LIN {X 0,Y 206.357,Z 449.351,A -85,B 0,C 180,E1 -22994.34,E2 -22994.34} C_VEL
LIN {X 0,Y 205.229,Z 439.622,A -85,B 0,C 180,E1 -22997.247,E2 -22997.247} C_VEL
LIN {X 0,Y 203.64,Z 431.973,A -85,B 0,C 180,E1 -22999.611,E2 -22999.611} C_VEL
LIN {X 0,Y 201.242,Z 425.032,A -85,B 0,C 180,E1 -23002.05,E2 -23002.05} C_VEL
LIN {X 0,Y 197.447,Z 417.118,A -85,B 0,C 180,E1 -23005.284,E2 -23005.284} C_VEL
LIN {X 0,Y 193.926,Z 410.394,A -85,B 0,C 180,E1 -23008.299,E2 -23008.299} C_VEL
LIN {X 0,Y 191.536,Z 406.308,A -85,B 0,C 180,E1 -23010.369,E2 -23010.369} C_VEL
LIN {X 0,Y 189.131,Z 402.897,A -85,B 0,C 180,E1 -23012.398,E2 -23012.398} C_VEL
LIN {X 0,Y 188.252,Z 401.374,A -85,B 0,C 180,E1 -23013.235,E2 -23013.235} C_VEL
LIN {X 0,Y 185.97,Z 398.361,A -85,B 0,C 180,E1 -23015.354,E2 -23015.354} C_VEL
LIN {X 0,Y 185.027,Z 396.629,A -85,B 0,C 180,E1 -23016.346,E2 -23016.346} C_VEL
LIN {X 0,Y 182.514,Z 394.01,A -85,B 0,C 180,E1 -23018.838,E2 -23018.838} C_VEL
LIN {X 0,Y 181.303,Z 391.376,A -85,B 0,C 180,E1 -23020.467,E2 -23020.467} C_VEL
LIN {X 0,Y 178.541,Z 389.25,A -85,B 0,C 180,E1 -23023.712,E2 -23023.712} C_VEL
LIN {X 0,Y 177.229,Z 386.47,A -85,B 0,C 180,E1 -23026.016,E2 -23026.016} C_VEL
LIN {X 0,Y 177.02,Z 385.707,A -85,B 0,C 180,E1 -23026.511,E2 -23026.511} C_VEL
LIN {X 0,Y 172.999,Z 381.886,A -85,B 0,C 180,E1 -23040,E2 -23040} C_VEL
LIN {X 0,Y 174.879,Z 384.888,A -85,B 0,C 180,E1 -23048.959,E2 -23048.959} C_VEL
LIN {X 0,Y 177.427,Z 387.578,A -85,B 0,C 180,E1 -23053.602,E2 -23053.602} C_VEL
LIN {X 0,Y 179.019,Z 391.368,A -85,B 0,C 180,E1 -23056.243,E2 -23056.243} C_VEL
LIN {X 0,Y 181.998,Z 394.906,A -85,B 0,C 180,E1 -23059.748,E2 -23059.748} C_VEL
LIN {X 0,Y 183.712,Z 398.579,A -85,B 0,C 180,E1 -23061.752,E2 -23061.752} C_VEL
LIN {X 0,Y 185.943,Z 401.558,A -85,B 0,C 180,E1 -23063.899,E2 -23063.899} C_VEL
LIN {X 0,Y 187.812,Z 405.564,A -85,B 0,C 180,E1 -23065.786,E2 -23065.786} C_VEL
LIN {X 0,Y 189.272,Z 407.823,A -85,B 0,C 180,E1 -23067.048,E2 -23067.048} C_VEL
LIN {X 0,Y 191.444,Z 412.238,A -85,B 0,C 180,E1 -23069.03,E2 -23069.03} C_VEL
LIN {X 0,Y 194.937,Z 419.942,A -85,B 0,C 180,E1 -23072.125,E2 -23072.125} C_VEL
LIN {X 0,Y 197.223,Z 425.43,A -85,B 0,C 180,E1 -23074.142,E2 -23074.142} C_VEL
LIN {X 0,Y 200.62,Z 435.333,A -85,B 0,C 180,E1 -23077.407,E2 -23077.407} C_VEL
LIN {X 0,Y 201.683,Z 440.477,A -85,B 0,C 180,E1 -23078.847,E2 -23078.847} C_VEL
LIN {X 0,Y 202.508,Z 450.041,A -85,B 0,C 180,E1 -23081.253,E2 -23081.253} C_VEL
LIN {X 0,Y 202.585,Z 459.199,A -85,B 0,C 180,E1 -23083.502,E2 -23083.502} C_VEL
LIN {X 0,Y 201.927,Z 468.704,A -85,B 0,C 180,E1 -23085.887,E2 -23085.887} C_VEL
LIN {X 0,Y 200.829,Z 476.69,A -85,B 0,C 180,E1 -23087.965,E2 -23087.965} C_VEL
LIN {X 0,Y 195.602,Z 487.568,A -85,B 0,C 180,E1 -23090.376,E2 -23090.376} C_VEL
LIN {X 0,Y 190.484,Z 497.578,A -85,B 0,C 180,E1 -23093.163,E2 -23093.163} C_VEL
LIN {X 0,Y 185.183,Z 507.379,A -85,B 0,C 180,E1 -23096.609,E2 -23096.609} C_VEL
LIN {X 0,Y 180.687,Z 515.593,A -85,B 0,C 180,E1 -23100.271,E2 -23100.271} C_VEL
LIN {X 0,Y 176.716,Z 522.382,A -85,B 0,C 180,E1 -23104.059,E2 -23104.059} C_VEL
LIN {X 0,Y 173.038,Z 529.281,A -85,B 0,C 180,E1 -23109.091,E2 -23109.091} C_VEL
LIN {X 0,Y 170.943,Z 533.56,A -85,B 0,C 180,E1 -23113.275,E2 -23113.275} C_VEL
LIN {X 0,Y 169.503,Z 537.155,A -85,B 0,C 180,E1 -23118.036,E2 -23118.036} C_VEL
LIN {X 0,Y 169.009,Z 539.54,A -85,B 0,C 180,E1 -23122.835,E2 -23122.835} C_VEL
LIN {X 0,Y 169.061,Z 540.479,A -85,B 0,C 180,E1 -23126.109,E2 -23126.109} C_VEL
LIN {X 0,Y 169.248,Z 540.917,A -85,B 0,C 180,E1 -23130.001,E2 -23130.001} C_VEL
LIN {X 0,Y 169.056,Z 540.278,A -85,B 0,C 180,E1 -23134.77,E2 -23134.77} C_VEL
LIN {X 0,Y 169.154,Z 538.458,A -85,B 0,C 180,E1 -23139.567,E2 -23139.567} C_VEL
LIN {X 0,Y 169.375,Z 537.495,A -85,B 0,C 180,E1 -23141.282,E2 -23141.282} C_VEL
LIN {X 0,Y 169.115,Z 536.308,A -85,B 0,C 180,E1 -23143.24,E2 -23143.24} C_VEL
LIN {X 0,Y 167.216,Z 533.952,A -85,B 0,C 180,E1 -23146.464,E2 -23146.464} C_VEL
LIN {X 0,Y 165.895,Z 531.695,A -85,B 0,C 180,E1 -23149.055,E2 -23149.055} C_VEL
LIN {X 0,Y 165.906,Z 529.739,A -85,B 0,C 180,E1 -23150.989,E2 -23150.989} C_VEL
LIN {X 0,Y 166.215,Z 529.037,A -85,B 0,C 180,E1 -23151.617,E2 -23151.617} C_VEL
LIN {X 0,Y 169.271,Z 523.624,A -85,B 0,C 180,E1 -23155.847,E2 -23155.847} C_VEL
LIN {X 0,Y 173.849,Z 516.138,A -85,B 0,C 180,E1 -23160.354,E2 -23160.354} C_VEL
LIN {X 0,Y 177.837,Z 509.382,A -85,B 0,C 180,E1 -23163.593,E2 -23163.593} C_VEL
LIN {X 0,Y 183.114,Z 500.046,A -85,B 0,C 180,E1 -23167.193,E2 -23167.193} C_VEL
LIN {X 0,Y 188.347,Z 490.582,A -85,B 0,C 180,E1 -23170.067,E2 -23170.067} C_VEL
LIN {X 0,Y 194.056,Z 479.351,A -85,B 0,C 180,E1 -23172.771,E2 -23172.771} C_VEL
LIN {X 0,Y 195.076,Z 476.407,A -85,B 0,C 180,E1 -23173.465,E2 -23173.465} C_VEL
LIN {X 0,Y 196.535,Z 465.476,A -85,B 0,C 180,E1 -23176.42,E2 -23176.42} C_VEL
LIN {X 0,Y 197.004,Z 454.416,A -85,B 0,C 180,E1 -23179.295,E2 -23179.295} C_VEL
LIN {X 0,Y 196.407,Z 443.528,A -85,B 0,C 180,E1 -23182.193,E2 -23182.193} C_VEL
LIN {X 0,Y 195.356,Z 438.125,A -85,B 0,C 180,E1 -23183.845,E2 -23183.845} C_VEL
LIN {X 0,Y 192.243,Z 428.566,A -85,B 0,C 180,E1 -23187.229,E2 -23187.229} C_VEL
LIN {X 0,Y 189.538,Z 421.776,A -85,B 0,C 180,E1 -23189.962,E2 -23189.962} C_VEL
LIN {X 0,Y 187.417,Z 417.073,A -85,B 0,C 180,E1 -23192.048,E2 -23192.048} C_VEL
LIN {X 0,Y 185.403,Z 412.52,A -85,B 0,C 180,E1 -23194.177,E2 -23194.177} C_VEL
LIN {X 0,Y 183.355,Z 408.488,A -85,B 0,C 180,E1 -23196.343,E2 -23196.343} C_VEL
LIN {X 0,Y 182.725,Z 407.139,A -85,B 0,C 180,E1 -23197.081,E2 -23197.081} C_VEL
LIN {X 0,Y 180.343,Z 403.371,A -85,B 0,C 180,E1 -23199.706,E2 -23199.706} C_VEL
LIN {X 0,Y 179.32,Z 400.892,A -85,B 0,C 180,E1 -23201.135,E2 -23201.135} C_VEL
LIN {X 0,Y 176.635,Z 397.089,A -85,B 0,C 180,E1 -23204.79,E2 -23204.79} C_VEL
LIN {X 0,Y 175.579,Z 394.08,A -85,B 0,C 180,E1 -23206.841,E2 -23206.841} C_VEL
LIN {X 0,Y 172.61,Z 390.708,A -85,B 0,C 180,E1 -23213.278,E2 -23213.278} C_VEL
LIN {X 0,Y 171.67,Z 388.393,A -85,B 0,C 180,E1 -23220,E2 -23220} C_VEL
LIN {X 0,Y 175.323,Z 392.776,A -85,B 0,C 180,E1 -23233.585,E2 -23233.585} C_VEL
LIN {X 0,Y 176.409,Z 395.611,A -85,B 0,C 180,E1 -23235.896,E2 -23235.896} C_VEL
LIN {X 0,Y 178.925,Z 397.987,A -85,B 0,C 180,E1 -23239.207,E2 -23239.207} C_VEL
LIN {X 0,Y 181.096,Z 401.825,A -85,B 0,C 180,E1 -23242.084,E2 -23242.084} C_VEL
LIN {X 0,Y 182.75,Z 403.698,A -85,B 0,C 180,E1 -23243.816,E2 -23243.816} C_VEL
LIN {X 0,Y 185.765,Z 408.54,A -85,B 0,C 180,E1 -23247,E2 -23247} C_VEL
LIN {X 0,Y 188.461,Z 413.028,A -85,B 0,C 180,E1 -23249.612,E2 -23249.612} C_VEL
LIN {X 0,Y 192.28,Z 420.206,A -85,B 0,C 180,E1 -23253.248,E2 -23253.248} C_VEL
LIN {X 0,Y 196.021,Z 428.537,A -85,B 0,C 180,E1 -23256.909,E2 -23256.909} C_VEL
LIN {X 0,Y 198.377,Z 435.704,A -85,B 0,C 180,E1 -23259.621,E2 -23259.621} C_VEL
LIN {X 0,Y 199.887,Z 444.192,A -85,B 0,C 180,E1 -23262.407,E2 -23262.407} C_VEL
LIN {X 0,Y 200.624,Z 454.153,A -85,B 0,C 180,E1 -23265.523,E2 -23265.523} C_VEL
LIN {X 0,Y 200.457,Z 456.426,A -85,B 0,C 180,E1 -23266.176,E2 -23266.176} C_VEL
LIN {X 0,Y 195.569,Z 467.034,A -85,B 0,C 180,E1 -23268.331,E2 -23268.331} C_VEL
LIN {X 0,Y 190.126,Z 477.796,A -85,B 0,C 180,E1 -23271.066,E2 -23271.066} C_VEL
LIN {X 0,Y 185.207,Z 486.911,A -85,B 0,C 180,E1 -23273.971,E2 -23273.971} C_VEL
LIN {X 0,Y 179.891,Z 495.825,A -85,B 0,C 180,E1 -23277.507,E2 -23277.507} C_VEL
LIN {X 0,Y 175.25,Z 503.202,A -85,B 0,C 180,E1 -23281.233,E2 -23281.233} C_VEL
LIN {X 0,Y 170.88,Z 510.082,A -85,B 0,C 180,E1 -23285.714,E2 -23285.714} C_VEL
LIN {X 0,Y 167.33,Z 515.481,A -85,B 0,C 180,E1 -23290.365,E2 -23290.365} C_VEL
LIN {X 0,Y 164.88,Z 519.538,A -85,B 0,C 180,E1 -23295.181,E2 -23295.181} C_VEL
LIN {X 0,Y 163.213,Z 522.382,A -85,B 0,C 180,E1 -23300.081,E2 -23300.081} C_VEL
LIN {X 0,Y 162.448,Z 524.08,A -85,B 0,C 180,E1 -23305.035,E2 -23305.035} C_VEL
LIN {X 0,Y 162.264,Z 524.667,A -85,B 0,C 180,E1 -23309.999,E2 -23309.999} C_VEL
LIN {X 0,Y 162.431,Z 524.114,A -85,B 0,C 180,E1 -23314.963,E2 -23314.963} C_VEL
LIN {X 0,Y 163.21,Z 522.46,A -85,B 0,C 180,E1 -23319.917,E2 -23319.917} C_VEL
LIN {X 0,Y 164.838,Z 519.657,A -85,B 0,C 180,E1 -23324.821,E2 -23324.821} C_VEL
LIN {X 0,Y 167.276,Z 515.639,A -85,B 0,C 180,E1 -23329.639,E2 -23329.639} C_VEL
LIN {X 0,Y 170.797,Z 510.291,A -85,B 0,C 180,E1 -23334.297,E2 -23334.297} C_VEL
LIN {X 0,Y 173.967,Z 505.297,A -85,B 0,C 180,E1 -23337.682,E2 -23337.682} C_VEL
LIN {X 0,Y 178.452,Z 498.328,A -85,B 0,C 180,E1 -23341.454,E2 -23341.454} C_VEL
LIN {X 0,Y 183.49,Z 489.94,A -85,B 0,C 180,E1 -23345.065,E2 -23345.065} C_VEL
LIN {X 0,Y 189.161,Z 479.921,A -85,B 0,C 180,E1 -23348.443,E2 -23348.443} C_VEL
LIN {X 0,Y 193.577,Z 471.337,A -85,B 0,C 180,E1 -23350.805,E2 -23350.805} C_VEL
LIN {X 0,Y 199.392,Z 459.291,A -85,B 0,C 180,E1 -23353.417,E2 -23353.417} C_VEL
LIN {X 0,Y 200.718,Z 455.857,A -85,B 0,C 180,E1 -23354.098,E2 -23354.098} C_VEL
LIN {X 0,Y 200.295,Z 447.148,A -85,B 0,C 180,E1 -23356.827,E2 -23356.827} C_VEL
LIN {X 0,Y 198.949,Z 437.956,A -85,B 0,C 180,E1 -23359.788,E2 -23359.788} C_VEL
LIN {X 0,Y 197.316,Z 431.708,A -85,B 0,C 180,E1 -23362.001,E2 -23362.001} C_VEL
LIN {X 0,Y 194.078,Z 424.015,A -85,B 0,C 180,E1 -23365.226,E2 -23365.226} C_VEL
LIN {X 0,Y 190.313,Z 416.234,A -85,B 0,C 180,E1 -23368.868,E2 -23368.868} C_VEL
LIN {X 0,Y 188.189,Z 412.289,A -85,B 0,C 180,E1 -23370.955,E2 -23370.955} C_VEL
LIN {X 0,Y 182.602,Z 403.311,A -85,B 0,C 180,E1 -23376.69,E2 -23376.69} C_VEL
LIN {X 0,Y 179.966,Z 400.122,A -85,B 0,C 180,E1 -23379.664,E2 -23379.664} C_VEL
LIN {X 0,Y 179.04,Z 398.02,A -85,B 0,C 180,E1 -23381.045,E2 -23381.045} C_VEL
LIN {X 0,Y 176.502,Z 395.71,A -85,B 0,C 180,E1 -23384.408,E2 -23384.408} C_VEL
LIN {X 0,Y 175.352,Z 392.774,A -85,B 0,C 180,E1 -23386.897,E2 -23386.897} C_VEL
LIN {X 0,Y 171.894,Z 388.908,A -85,B 0,C 180,E1 -23400,E2 -23400} C_VEL
LIN {X 0,Y 173.577,Z 391.852,A -85,B 0,C 180,E1 -23408.733,E2 -23408.733} C_VEL
LIN {X 0,Y 175.707,Z 394.352,A -85,B 0,C 180,E1 -23413.002,E2 -23413.002} C_VEL
LIN {X 0,Y 177.14,Z 397.978,A -85,B 0,C 180,E1 -23415.681,E2 -23415.681} C_VEL
LIN {X 0,Y 179.687,Z 401.392,A -85,B 0,C 180,E1 -23419.047,E2 -23419.047} C_VEL
LIN {X 0,Y 181.35,Z 405.086,A -85,B 0,C 180,E1 -23421.229,E2 -23421.229} C_VEL
LIN {X 0,Y 183.161,Z 407.746,A -85,B 0,C 180,E1 -23423.16,E2 -23423.16} C_VEL
LIN {X 0,Y 185.034,Z 411.929,A -85,B 0,C 180,E1 -23425.296,E2 -23425.296} C_VEL
LIN {X 0,Y 186.069,Z 413.773,A -85,B 0,C 180,E1 -23426.302,E2 -23426.302} C_VEL
LIN {X 0,Y 188.643,Z 419.492,A -85,B 0,C 180,E1 -23428.968,E2 -23428.968} C_VEL
LIN {X 0,Y 192.315,Z 428.597,A -85,B 0,C 180,E1 -23432.68,E2 -23432.68} C_VEL
LIN {X 0,Y 195.584,Z 438.822,A -85,B 0,C 180,E1 -23436.293,E2 -23436.293} C_VEL
LIN {X 0,Y 196.691,Z 445.183,A -85,B 0,C 180,E1 -23438.18,E2 -23438.18} C_VEL
LIN {X 0,Y 197.085,Z 455.509,A -85,B 0,C 180,E1 -23440.925,E2 -23440.925} C_VEL
LIN {X 0,Y 196.495,Z 467.003,A -85,B 0,C 180,E1 -23443.929,E2 -23443.929} C_VEL
LIN {X 0,Y 194.961,Z 477.492,A -85,B 0,C 180,E1 -23446.772,E2 -23446.772} C_VEL
LIN {X 0,Y 189.232,Z 489.017,A -85,B 0,C 180,E1 -23449.464,E2 -23449.464} C_VEL
LIN {X 0,Y 183.939,Z 498.727,A -85,B 0,C 180,E1 -23452.315,E2 -23452.315} C_VEL
LIN {X 0,Y 178.827,Z 507.692,A -85,B 0,C 180,E1 -23455.62,E2 -23455.62} C_VEL
LIN {X 0,Y 173.865,Z 516.266,A -85,B 0,C 180,E1 -23459.651,E2 -23459.651} C_VEL
LIN {X 0,Y 169.271,Z 523.722,A -85,B 0,C 180,E1 -23464.155,E2 -23464.155} C_VEL
LIN {X 0,Y 166.142,Z 529.276,A -85,B 0,C 180,E1 -23468.532,E2 -23468.532} C_VEL
LIN {X 0,Y 164.064,Z 533.208,A -85,B 0,C 180,E1 -23472.552,E2 -23472.552} C_VEL
LIN {X 0,Y 162.498,Z 536.804,A -85,B 0,C 180,E1 -23477.512,E2 -23477.512} C_VEL
LIN {X 0,Y 161.924,Z 539.19,A -85,B 0,C 180,E1 -23482.519,E2 -23482.519} C_VEL
LIN {X 0,Y 161.964,Z 540.222,A -85,B 0,C 180,E1 -23486.393,E2 -23486.393} C_VEL
LIN {X 0,Y 162.167,Z 540.57,A -85,B 0,C 180,E1 -23490.001,E2 -23490.001} C_VEL
LIN {X 0,Y 161.946,Z 539.928,A -85,B 0,C 180,E1 -23494.98,E2 -23494.98} C_VEL
LIN {X 0,Y 162.107,Z 538.107,A -85,B 0,C 180,E1 -23499.988,E2 -23499.988} C_VEL
LIN {X 0,Y 163.137,Z 535.106,A -85,B 0,C 180,E1 -23504.981,E2 -23504.981} C_VEL
LIN {X 0,Y 165.255,Z 530.865,A -85,B 0,C 180,E1 -23509.892,E2 -23509.892} C_VEL
LIN {X 0,Y 166.215,Z 529.037,A -85,B 0,C 180,E1 -23511.617,E2 -23511.617} C_VEL
LIN {X 0,Y 166.827,Z 526.887,A -85,B 0,C 180,E1 -23513.493,E2 -23513.493} C_VEL
LIN {X 0,Y 166.204,Z 519.756,A -85,B 0,C 180,E1 -23519.123,E2 -23519.123} C_VEL
LIN {X 0,Y 166.985,Z 517.012,A -85,B 0,C 180,E1 -23520.904,E2 -23520.904} C_VEL
LIN {X 0,Y 167.525,Z 516.025,A -85,B 0,C 180,E1 -23521.462,E2 -23521.462} C_VEL
LIN {X 0,Y 172.577,Z 507.794,A -85,B 0,C 180,E1 -23525.465,E2 -23525.465} C_VEL
LIN {X 0,Y 178.346,Z 498.194,A -85,B 0,C 180,E1 -23529.089,E2 -23529.089} C_VEL
LIN {X 0,Y 183.836,Z 488.443,A -85,B 0,C 180,E1 -23531.993,E2 -23531.993} C_VEL
LIN {X 0,Y 188.881,Z 478.998,A -85,B 0,C 180,E1 -23534.241,E2 -23534.241} C_VEL
LIN {X 0,Y 190.432,Z 470.051,A -85,B 0,C 180,E1 -23536.793,E2 -23536.793} C_VEL
LIN {X 0,Y 191.405,Z 460.211,A -85,B 0,C 180,E1 -23539.513,E2 -23539.513} C_VEL
LIN {X 0,Y 191.437,Z 449.894,A -85,B 0,C 180,E1 -23542.387,E2 -23542.387} C_VEL
LIN {X 0,Y 190.929,Z 444.234,A -85,B 0,C 180,E1 -23544.079,E2 -23544.079} C_VEL
LIN {X 0,Y 188.11,Z 434.077,A -85,B 0,C 180,E1 -23547.817,E2 -23547.817} C_VEL
LIN {X 0,Y 185.33,Z 426.351,A -85,B 0,C 180,E1 -23551.086,E2 -23551.086} C_VEL
LIN {X 0,Y 182.601,Z 419.461,A -85,B 0,C 180,E1 -23554.343,E2 -23554.343} C_VEL
LIN {X 0,Y 179.328,Z 412.591,A -85,B 0,C 180,E1 -23558.333,E2 -23558.333} C_VEL
LIN {X 0,Y 177.226,Z 408.252,A -85,B 0,C 180,E1 -23561.204,E2 -23561.204} C_VEL
LIN {X 0,Y 176.746,Z 407.099,A -85,B 0,C 180,E1 -23561.977,E2 -23561.977} C_VEL
LIN {X 0,Y 174.423,Z 403.409,A -85,B 0,C 180,E1 -23565.554,E2 -23565.554} C_VEL
LIN {X 0,Y 173.633,Z 400.759,A -85,B 0,C 180,E1 -23567.435,E2 -23567.435} C_VEL
LIN {X 0,Y 171.059,Z 397.556,A -85,B 0,C 180,E1 -23573.661,E2 -23573.661} C_VEL
LIN {X 0,Y 170.307,Z 395.372,A -85,B 0,C 180,E1 -23580,E2 -23580} C_VEL
LIN {X 0,Y 173.338,Z 399.597,A -85,B 0,C 180,E1 -23593.115,E2 -23593.115} C_VEL
LIN {X 0,Y 174.397,Z 402.424,A -85,B 0,C 180,E1 -23595.635,E2 -23595.635} C_VEL
LIN {X 0,Y 176.681,Z 404.826,A -85,B 0,C 180,E1 -23598.955,E2 -23598.955} C_VEL
LIN {X 0,Y 177.884,Z 407.4,A -85,B 0,C 180,E1 -23600.829,E2 -23600.829} C_VEL
LIN {X 0,Y 179.705,Z 409.616,A -85,B 0,C 180,E1 -23603.022,E2 -23603.022} C_VEL
LIN {X 0,Y 182.445,Z 414.39,A -85,B 0,C 180,E1 -23606.295,E2 -23606.295} C_VEL
LIN {X 0,Y 185.331,Z 419.821,A -85,B 0,C 180,E1 -23609.537,E2 -23609.537} C_VEL
LIN {X 0,Y 188.386,Z 426.072,A -85,B 0,C 180,E1 -23612.839,E2 -23612.839} C_VEL
LIN {X 0,Y 191.66,Z 434.084,A -85,B 0,C 180,E1 -23616.509,E2 -23616.509} C_VEL
LIN {X 0,Y 193.437,Z 440.358,A -85,B 0,C 180,E1 -23618.992,E2 -23618.992} C_VEL
LIN {X 0,Y 194.566,Z 448.821,A -85,B 0,C 180,E1 -23621.932,E2 -23621.932} C_VEL
LIN {X 0,Y 194.864,Z 458.05,A -85,B 0,C 180,E1 -23624.977,E2 -23624.977} C_VEL
LIN {X 0,Y 189.36,Z 469.319,A -85,B 0,C 180,E1 -23627.363,E2 -23627.363} C_VEL
LIN {X 0,Y 184.633,Z 478.149,A -85,B 0,C 180,E1 -23629.675,E2 -23629.675} C_VEL
LIN {X 0,Y 179.507,Z 487.261,A -85,B 0,C 180,E1 -23632.637,E2 -23632.637} C_VEL
LIN {X 0,Y 173.941,Z 496.175,A -85,B 0,C 180,E1 -23636.249,E2 -23636.249} C_VEL
LIN {X 0,Y 169.059,Z 503.552,A -85,B 0,C 180,E1 -23640.075,E2 -23640.075} C_VEL
LIN {X 0,Y 164.39,Z 510.433,A -85,B 0,C 180,E1 -23644.689,E2 -23644.689} C_VEL
LIN {X 0,Y 160.641,Z 515.831,A -85,B 0,C 180,E1 -23649.512,E2 -23649.512} C_VEL
LIN {X 0,Y 158.001,Z 519.888,A -85,B 0,C 180,E1 -23654.52,E2 -23654.52} C_VEL
LIN {X 0,Y 156.234,Z 522.73,A -85,B 0,C 180,E1 -23659.633,E2 -23659.633} C_VEL
LIN {X 0,Y 155.383,Z 524.427,A -85,B 0,C 180,E1 -23664.809,E2 -23664.809} C_VEL
LIN {X 0,Y 155.187,Z 525.014,A -85,B 0,C 180,E1 -23669.999,E2 -23669.999} C_VEL
LIN {X 0,Y 155.473,Z 524.299,A -85,B 0,C 180,E1 -23676.015,E2 -23676.015} C_VEL
LIN {X 0,Y 156.229,Z 522.807,A -85,B 0,C 180,E1 -23680.365,E2 -23680.365} C_VEL
LIN {X 0,Y 157.962,Z 520.006,A -85,B 0,C 180,E1 -23685.482,E2 -23685.482} C_VEL
LIN {X 0,Y 160.586,Z 515.987,A -85,B 0,C 180,E1 -23690.493,E2 -23690.493} C_VEL
LIN {X 0,Y 164.297,Z 510.641,A -85,B 0,C 180,E1 -23695.324,E2 -23695.324} C_VEL
LIN {X 0,Y 168.968,Z 503.817,A -85,B 0,C 180,E1 -23699.941,E2 -23699.941} C_VEL
LIN {X 0,Y 173.858,Z 496.471,A -85,B 0,C 180,E1 -23703.767,E2 -23703.767} C_VEL
LIN {X 0,Y 179.384,Z 487.606,A -85,B 0,C 180,E1 -23707.391,E2 -23707.391} C_VEL
LIN {X 0,Y 184.809,Z 478.087,A -85,B 0,C 180,E1 -23710.485,E2 -23710.485} C_VEL
LIN {X 0,Y 190.215,Z 467.874,A -85,B 0,C 180,E1 -23713.119,E2 -23713.119} C_VEL
LIN {X 0,Y 194.774,Z 458.524,A -85,B 0,C 180,E1 -23715.081,E2 -23715.081} C_VEL
LIN {X 0,Y 194.957,Z 455.123,A -85,B 0,C 180,E1 -23716.134,E2 -23716.134} C_VEL
LIN {X 0,Y 194.521,Z 447.32,A -85,B 0,C 180,E1 -23718.748,E2 -23718.748} C_VEL
LIN {X 0,Y 193.512,Z 440.125,A -85,B 0,C 180,E1 -23721.25,E2 -23721.25} C_VEL
LIN {X 0,Y 191.645,Z 433.849,A -85,B 0,C 180,E1 -23723.781,E2 -23723.781} C_VEL
LIN {X 0,Y 188.336,Z 425.795,A -85,B 0,C 180,E1 -23727.494,E2 -23727.494} C_VEL
LIN {X 0,Y 184.709,Z 418.303,A -85,B 0,C 180,E1 -23731.477,E2 -23731.477} C_VEL
LIN {X 0,Y 179.918,Z 410.036,A -85,B 0,C 180,E1 -23737.007,E2 -23737.007} C_VEL
LIN {X 0,Y 177.081,Z 405.761,A -85,B 0,C 180,E1 -23740.75,E2 -23740.75} C_VEL
LIN {X 0,Y 176.487,Z 404.509,A -85,B 0,C 180,E1 -23741.724,E2 -23741.724} C_VEL
LIN {X 0,Y 174.163,Z 401.948,A -85,B 0,C 180,E1 -23745.317,E2 -23745.317} C_VEL
LIN {X 0,Y 173.237,Z 399.316,A -85,B 0,C 180,E1 -23747.702,E2 -23747.702} C_VEL
LIN {X 0,Y 170.505,Z 395.884,A -85,B 0,C 180,E1 -23760,E2 -23760} C_VEL
LIN {X 0,Y 172.004,Z 398.75,A -85,B 0,C 180,E1 -23768.517,E2 -23768.517} C_VEL
LIN {X 0,Y 173.753,Z 401.032,A -85,B 0,C 180,E1 -23772.408,E2 -23772.408} C_VEL
LIN {X 0,Y 175.18,Z 404.84,A -85,B 0,C 180,E1 -23775.413,E2 -23775.413} C_VEL
LIN {X 0,Y 177.216,Z 407.877,A -85,B 0,C 180,E1 -23778.415,E2 -23778.415} C_VEL
LIN {X 0,Y 178.944,Z 411.83,A -85,B 0,C 180,E1 -23780.951,E2 -23780.951} C_VEL
LIN {X 0,Y 180.106,Z 413.513,A -85,B 0,C 180,E1 -23782.263,E2 -23782.263} C_VEL
LIN {X 0,Y 181.329,Z 416.899,A -85,B 0,C 180,E1 -23784.014,E2 -23784.014} C_VEL
LIN {X 0,Y 182.745,Z 419.751,A -85,B 0,C 180,E1 -23785.636,E2 -23785.636} C_VEL
LIN {X 0,Y 185.022,Z 425.348,A -85,B 0,C 180,E1 -23788.347,E2 -23788.347} C_VEL
LIN {X 0,Y 187.793,Z 432.86,A -85,B 0,C 180,E1 -23791.597,E2 -23791.597} C_VEL
LIN {X 0,Y 190.354,Z 441.59,A -85,B 0,C 180,E1 -23794.91,E2 -23794.91} C_VEL
LIN {X 0,Y 191.353,Z 446.787,A -85,B 0,C 180,E1 -23796.643,E2 -23796.643} C_VEL
LIN {X 0,Y 191.618,Z 455.971,A -85,B 0,C 180,E1 -23799.248,E2 -23799.248} C_VEL
LIN {X 0,Y 191.217,Z 463.853,A -85,B 0,C 180,E1 -23801.42,E2 -23801.42} C_VEL
LIN {X 0,Y 189.973,Z 473.824,A -85,B 0,C 180,E1 -23804.214,E2 -23804.214} C_VEL
LIN {X 0,Y 188.896,Z 479.242,A -85,B 0,C 180,E1 -23805.766,E2 -23805.766} C_VEL
LIN {X 0,Y 182.905,Z 490.439,A -85,B 0,C 180,E1 -23808.486,E2 -23808.486} C_VEL
LIN {X 0,Y 176.582,Z 501.319,A -85,B 0,C 180,E1 -23811.911,E2 -23811.911} C_VEL
LIN {X 0,Y 171.15,Z 510.407,A -85,B 0,C 180,E1 -23815.625,E2 -23815.625} C_VEL
LIN {X 0,Y 166.37,Z 517.957,A -85,B 0,C 180,E1 -23819.542,E2 -23819.542} C_VEL
LIN {X 0,Y 161.834,Z 525.012,A -85,B 0,C 180,E1 -23824.262,E2 -23824.262} C_VEL
LIN {X 0,Y 158.495,Z 530.582,A -85,B 0,C 180,E1 -23829.224,E2 -23829.224} C_VEL
LIN {X 0,Y 156.226,Z 534.81,A -85,B 0,C 180,E1 -23834.342,E2 -23834.342} C_VEL
LIN {X 0,Y 155.041,Z 537.794,A -85,B 0,C 180,E1 -23839.554,E2 -23839.554} C_VEL
LIN {X 0,Y 154.846,Z 539.595,A -85,B 0,C 180,E1 -23844.793,E2 -23844.793} C_VEL
LIN {X 0,Y 155.067,Z 540.222,A -85,B 0,C 180,E1 -23850.001,E2 -23850.001} C_VEL
LIN {X 0,Y 154.848,Z 539.578,A -85,B 0,C 180,E1 -23855.209,E2 -23855.209} C_VEL
LIN {X 0,Y 155.08,Z 537.757,A -85,B 0,C 180,E1 -23860.445,E2 -23860.445} C_VEL
LIN {X 0,Y 156.23,Z 534.754,A -85,B 0,C 180,E1 -23865.66,E2 -23865.66} C_VEL
LIN {X 0,Y 158.513,Z 530.512,A -85,B 0,C 180,E1 -23870.776,E2 -23870.776} C_VEL
LIN {X 0,Y 161.836,Z 524.915,A -85,B 0,C 180,E1 -23875.74,E2 -23875.74} C_VEL
LIN {X 0,Y 166.36,Z 517.826,A -85,B 0,C 180,E1 -23880.462,E2 -23880.462} C_VEL
LIN {X 0,Y 167.525,Z 516.025,A -85,B 0,C 180,E1 -23881.462,E2 -23881.462} C_VEL
LIN {X 0,Y 168.808,Z 513.064,A -85,B 0,C 180,E1 -23883.151,E2 -23883.151} C_VEL
LIN {X 0,Y 169.476,Z 508.033,A -85,B 0,C 180,E1 -23886.044,E2 -23886.044} C_VEL
LIN {X 0,Y 170.473,Z 502.549,A -85,B 0,C 180,E1 -23888.805,E2 -23888.805} C_VEL
LIN {X 0,Y 172.2,Z 498.882,A -85,B 0,C 180,E1 -23890.236,E2 -23890.236} C_VEL
LIN {X 0,Y 178.579,Z 488.089,A -85,B 0,C 180,E1 -23893.53,E2 -23893.53} C_VEL
LIN {X 0,Y 183.148,Z 479.713,A -85,B 0,C 180,E1 -23895.583,E2 -23895.583} C_VEL
LIN {X 0,Y 185.063,Z 469.654,A -85,B 0,C 180,E1 -23898.595,E2 -23898.595} C_VEL
LIN {X 0,Y 186.126,Z 458.7,A -85,B 0,C 180,E1 -23901.809,E2 -23901.809} C_VEL
LIN {X 0,Y 186.115,Z 450.316,A -85,B 0,C 180,E1 -23904.322,E2 -23904.322} C_VEL
LIN {X 0,Y 185.318,Z 445.395,A -85,B 0,C 180,E1 -23906.076,E2 -23906.076} C_VEL
LIN {X 0,Y 183.162,Z 437.048,A -85,B 0,C 180,E1 -23909.442,E2 -23909.442} C_VEL
LIN {X 0,Y 180.314,Z 428.581,A -85,B 0,C 180,E1 -23913.371,E2 -23913.371} C_VEL
LIN {X 0,Y 178.706,Z 424.196,A -85,B 0,C 180,E1 -23915.611,E2 -23915.611} C_VEL
LIN {X 0,Y 176.317,Z 418.715,A -85,B 0,C 180,E1 -23918.977,E2 -23918.977} C_VEL
LIN {X 0,Y 174.82,Z 415.549,A -85,B 0,C 180,E1 -23921.24,E2 -23921.24} C_VEL
LIN {X 0,Y 174.285,Z 413.624,A -85,B 0,C 180,E1 -23922.396,E2 -23922.396} C_VEL
LIN {X 0,Y 172.099,Z 409.894,A -85,B 0,C 180,E1 -23926.119,E2 -23926.119} C_VEL
LIN {X 0,Y 171.375,Z 407.292,A -85,B 0,C 180,E1 -23928.168,E2 -23928.168} C_VEL
LIN {X 0,Y 169.237,Z 404.365,A -85,B 0,C 180,E1 -23934.041,E2 -23934.041} C_VEL
LIN {X 0,Y 168.643,Z 402.308,A -85,B 0,C 180,E1 -23940,E2 -23940} C_VEL
LIN {X 0,Y 171.102,Z 406.261,A -85,B 0,C 180,E1 -23952.604,E2 -23952.604} C_VEL
LIN {X 0,Y 171.64,Z 408.08,A -85,B 0,C 180,E1 -23954.222,E2 -23954.222} C_VEL
LIN {X 0,Y 174.187,Z 411.885,A -85,B 0,C 180,E1 -23958.831,E2 -23958.831} C_VEL
LIN {X 0,Y 176.494,Z 415.577,A -85,B 0,C 180,E1 -23962.228,E2 -23962.228} C_VEL
LIN {X 0,Y 178.939,Z 420.188,A -85,B 0,C 180,E1 -23965.597,E2 -23965.597} C_VEL
LIN {X 0,Y 182.473,Z 427.355,A -85,B 0,C 180,E1 -23970.046,E2 -23970.046} C_VEL
LIN {X 0,Y 185.964,Z 436.051,A -85,B 0,C 180,E1 -23974.534,E2 -23974.534} C_VEL
LIN {X 0,Y 187.598,Z 441.129,A -85,B 0,C 180,E1 -23976.828,E2 -23976.828} C_VEL
LIN {X 0,Y 188.689,Z 447.432,A -85,B 0,C 180,E1 -23979.286,E2 -23979.286} C_VEL
LIN {X 0,Y 189.182,Z 455.756,A -85,B 0,C 180,E1 -23982.289,E2 -23982.289} C_VEL
LIN {X 0,Y 189.071,Z 460.211,A -85,B 0,C 180,E1 -23983.817,E2 -23983.817} C_VEL
LIN {X 0,Y 183.204,Z 471.581,A -85,B 0,C 180,E1 -23986.328,E2 -23986.328} C_VEL
LIN {X 0,Y 178.003,Z 480.807,A -85,B 0,C 180,E1 -23988.924,E2 -23988.924} C_VEL
LIN {X 0,Y 172.148,Z 490.291,A -85,B 0,C 180,E1 -23992.237,E2 -23992.237} C_VEL
LIN {X 0,Y 166.549,Z 498.736,A -85,B 0,C 180,E1 -23996.004,E2 -23996.004} C_VEL
LIN {X 0,Y 161.585,Z 505.757,A -85,B 0,C 180,E1 -23999.987,E2 -23999.987} C_VEL
LIN {X 0,Y 156.932,Z 512.255,A -85,B 0,C 180,E1 -24004.82,E2 -24004.82} C_VEL
LIN {X 0,Y 153.199,Z 517.326,A -85,B 0,C 180,E1 -24009.874,E2 -24009.874} C_VEL
LIN {X 0,Y 151.156,Z 520.237,A -85,B 0,C 180,E1 -24013.8,E2 -24013.8} C_VEL
LIN {X 0,Y 149.24,Z 523.08,A -85,B 0,C 180,E1 -24019.141,E2 -24019.141} C_VEL
LIN {X 0,Y 148.325,Z 524.775,A -85,B 0,C 180,E1 -24024.561,E2 -24024.561} C_VEL
LIN {X 0,Y 148.112,Z 525.361,A -85,B 0,C 180,E1 -24029.999,E2 -24029.999} C_VEL
LIN {X 0,Y 148.369,Z 524.733,A -85,B 0,C 180,E1 -24035.88,E2 -24035.88} C_VEL
LIN {X 0,Y 149.233,Z 523.156,A -85,B 0,C 180,E1 -24040.857,E2 -24040.857} C_VEL
LIN {X 0,Y 151.117,Z 520.354,A -85,B 0,C 180,E1 -24046.202,E2 -24046.202} C_VEL
LIN {X 0,Y 153.938,Z 516.335,A -85,B 0,C 180,E1 -24051.421,E2 -24051.421} C_VEL
LIN {X 0,Y 157.871,Z 510.989,A -85,B 0,C 180,E1 -24056.433,E2 -24056.433} C_VEL
LIN {X 0,Y 162.839,Z 504.164,A -85,B 0,C 180,E1 -24061.191,E2 -24061.191} C_VEL
LIN {X 0,Y 168.781,Z 495.63,A -85,B 0,C 180,E1 -24065.657,E2 -24065.657} C_VEL
LIN {X 0,Y 174.717,Z 486.544,A -85,B 0,C 180,E1 -24069.311,E2 -24069.311} C_VEL
LIN {X 0,Y 180.124,Z 477.295,A -85,B 0,C 180,E1 -24072.302,E2 -24072.302} C_VEL
LIN {X 0,Y 186.169,Z 466.278,A -85,B 0,C 180,E1 -24075.057,E2 -24075.057} C_VEL
LIN {X 0,Y 189.006,Z 460.632,A -85,B 0,C 180,E1 -24076.238,E2 -24076.238} C_VEL
LIN {X 0,Y 189.293,Z 458.382,A -85,B 0,C 180,E1 -24076.951,E2 -24076.951} C_VEL
LIN {X 0,Y 189.106,Z 450.896,A -85,B 0,C 180,E1 -24079.594,E2 -24079.594} C_VEL
LIN {X 0,Y 188.402,Z 444.349,A -85,B 0,C 180,E1 -24082.01,E2 -24082.01} C_VEL
LIN {X 0,Y 186.982,Z 438.82,A -85,B 0,C 180,E1 -24084.367,E2 -24084.367} C_VEL
LIN {X 0,Y 183.967,Z 430.788,A -85,B 0,C 180,E1 -24088.312,E2 -24088.312} C_VEL
LIN {X 0,Y 180.904,Z 423.867,A -85,B 0,C 180,E1 -24092.212,E2 -24092.212} C_VEL
LIN {X 0,Y 177.428,Z 417.554,A -85,B 0,C 180,E1 -24096.665,E2 -24096.665} C_VEL
LIN {X 0,Y 176.701,Z 415.958,A -85,B 0,C 180,E1 -24097.799,E2 -24097.799} C_VEL
LIN {X 0,Y 173.794,Z 410.924,A -85,B 0,C 180,E1 -24102.344,E2 -24102.344} C_VEL
LIN {X 0,Y 171.85,Z 408.501,A -85,B 0,C 180,E1 -24105.796,E2 -24105.796} C_VEL
LIN {X 0,Y 171.07,Z 406.031,A -85,B 0,C 180,E1 -24108.146,E2 -24108.146} C_VEL
LIN {X 0,Y 168.832,Z 402.807,A -85,B 0,C 180,E1 -24120,E2 -24120} C_VEL
LIN {X 0,Y 170.163,Z 405.572,A -85,B 0,C 180,E1 -24128.311,E2 -24128.311} C_VEL
LIN {X 0,Y 171.571,Z 407.603,A -85,B 0,C 180,E1 -24131.818,E2 -24131.818} C_VEL
LIN {X 0,Y 172.862,Z 411.434,A -85,B 0,C 180,E1 -24135.012,E2 -24135.012} C_VEL
LIN {X 0,Y 174.451,Z 413.926,A -85,B 0,C 180,E1 -24137.586,E2 -24137.586} C_VEL
LIN {X 0,Y 175.707,Z 417.392,A -85,B 0,C 180,E1 -24139.876,E2 -24139.876} C_VEL
LIN {X 0,Y 176.538,Z 418.812,A -85,B 0,C 180,E1 -24140.995,E2 -24140.995} C_VEL
LIN {X 0,Y 179.236,Z 425.532,A -85,B 0,C 180,E1 -24144.93,E2 -24144.93} C_VEL
LIN {X 0,Y 181.244,Z 431.113,A -85,B 0,C 180,E1 -24147.73,E2 -24147.73} C_VEL
LIN {X 0,Y 184.042,Z 439.93,A -85,B 0,C 180,E1 -24151.673,E2 -24151.673} C_VEL
LIN {X 0,Y 185.981,Z 448.366,A -85,B 0,C 180,E1 -24154.944,E2 -24154.944} C_VEL
LIN {X 0,Y 186.319,Z 453.623,A -85,B 0,C 180,E1 -24156.622,E2 -24156.622} C_VEL
LIN {X 0,Y 185.883,Z 463.706,A -85,B 0,C 180,E1 -24159.6,E2 -24159.6} C_VEL
LIN {X 0,Y 184.526,Z 473.434,A -85,B 0,C 180,E1 -24162.446,E2 -24162.446} C_VEL
LIN {X 0,Y 183.214,Z 479.908,A -85,B 0,C 180,E1 -24164.418,E2 -24164.418} C_VEL
LIN {X 0,Y 177.598,Z 490.09,A -85,B 0,C 180,E1 -24166.952,E2 -24166.952} C_VEL
LIN {X 0,Y 170.993,Z 500.969,A -85,B 0,C 180,E1 -24170.428,E2 -24170.428} C_VEL
LIN {X 0,Y 165.255,Z 510.056,A -85,B 0,C 180,E1 -24174.215,E2 -24174.215} C_VEL
LIN {X 0,Y 160.25,Z 517.609,A -85,B 0,C 180,E1 -24178.247,E2 -24178.247} C_VEL
LIN {X 0,Y 155.381,Z 524.66,A -85,B 0,C 180,E1 -24183.109,E2 -24183.109} C_VEL
LIN {X 0,Y 151.795,Z 530.23,A -85,B 0,C 180,E1 -24188.261,E2 -24188.261} C_VEL
LIN {X 0,Y 149.346,Z 534.46,A -85,B 0,C 180,E1 -24193.601,E2 -24193.601} C_VEL
LIN {X 0,Y 148.009,Z 537.443,A -85,B 0,C 180,E1 -24199.052,E2 -24199.052} C_VEL
LIN {X 0,Y 147.736,Z 539.245,A -85,B 0,C 180,E1 -24204.542,E2 -24204.542} C_VEL
LIN {X 0,Y 147.823,Z 539.708,A -85,B 0,C 180,E1 -24207.276,E2 -24207.276} C_VEL
LIN {X 0,Y 147.971,Z 539.874,A -85,B 0,C 180,E1 -24210.001,E2 -24210.001} C_VEL
LIN {X 0,Y 147.818,Z 539.65,A -85,B 0,C 180,E1 -24213.201,E2 -24213.201} C_VEL
LIN {X 0,Y 147.776,Z 538.462,A -85,B 0,C 180,E1 -24218.204,E2 -24218.204} C_VEL
LIN {X 0,Y 148.518,Z 536.052,A -85,B 0,C 180,E1 -24223.687,E2 -24223.687} C_VEL
LIN {X 0,Y 150.424,Z 532.441,A -85,B 0,C 180,E1 -24229.091,E2 -24229.091} C_VEL
LIN {X 0,Y 153.457,Z 527.537,A -85,B 0,C 180,E1 -24234.343,E2 -24234.343} C_VEL
LIN {X 0,Y 157.614,Z 521.213,A -85,B 0,C 180,E1 -24239.374,E2 -24239.374} C_VEL
LIN {X 0,Y 162.305,Z 514.407,A -85,B 0,C 180,E1 -24243.512,E2 -24243.512} C_VEL
LIN {X 0,Y 167.431,Z 506.428,A -85,B 0,C 180,E1 -24247.341,E2 -24247.341} C_VEL
LIN {X 0,Y 172.2,Z 498.882,A -85,B 0,C 180,E1 -24250.236,E2 -24250.236} C_VEL
LIN {X 0,Y 174.135,Z 495.15,A -85,B 0,C 180,E1 -24251.578,E2 -24251.578} C_VEL
LIN {X 0,Y 176.011,Z 488.767,A -85,B 0,C 180,E1 -24253.964,E2 -24253.964} C_VEL
LIN {X 0,Y 178.091,Z 478.062,A -85,B 0,C 180,E1 -24257.792,E2 -24257.792} C_VEL
LIN {X 0,Y 179.778,Z 469.336,A -85,B 0,C 180,E1 -24260.512,E2 -24260.512} C_VEL
LIN {X 0,Y 180.778,Z 460.237,A -85,B 0,C 180,E1 -24263.334,E2 -24263.334} C_VEL
LIN {X 0,Y 180.896,Z 452.357,A -85,B 0,C 180,E1 -24265.896,E2 -24265.896} C_VEL
LIN {X 0,Y 179.033,Z 443.151,A -85,B 0,C 180,E1 -24269.727,E2 -24269.727} C_VEL
LIN {X 0,Y 176.774,Z 434.977,A -85,B 0,C 180,E1 -24273.596,E2 -24273.596} C_VEL
LIN {X 0,Y 175.116,Z 429.902,A -85,B 0,C 180,E1 -24276.339,E2 -24276.339} C_VEL
LIN {X 0,Y 173.01,Z 424.493,A -85,B 0,C 180,E1 -24279.801,E2 -24279.801} C_VEL
LIN {X 0,Y 171.253,Z 419.625,A -85,B 0,C 180,E1 -24283.306,E2 -24283.306} C_VEL
LIN {X 0,Y 169.493,Z 416.163,A -85,B 0,C 180,E1 -24286.818,E2 -24286.818} C_VEL
LIN {X 0,Y 169.143,Z 414.725,A -85,B 0,C 180,E1 -24288.01,E2 -24288.01} C_VEL
LIN {X 0,Y 168.317,Z 412.895,A -85,B 0,C 180,E1 -24290.386,E2 -24290.386} C_VEL
LIN {X 0,Y 166.991,Z 410.844,A -85,B 0,C 180,E1 -24295.172,E2 -24295.172} C_VEL
LIN {X 0,Y 166.686,Z 409.158,A -85,B 0,C 180,E1 -24300,E2 -24300} C_VEL
LIN {X 0,Y 168.643,Z 412.714,A -85,B 0,C 180,E1 -24312.027,E2 -24312.027} C_VEL
LIN {X 0,Y 169.36,Z 415.065,A -85,B 0,C 180,E1 -24314.418,E2 -24314.418} C_VEL
LIN {X 0,Y 171.073,Z 417.893,A -85,B 0,C 180,E1 -24317.946,E2 -24317.946} C_VEL
LIN {X 0,Y 173.117,Z 421.479,A -85,B 0,C 180,E1 -24321.431,E2 -24321.431} C_VEL
LIN {X 0,Y 175.235,Z 425.799,A -85,B 0,C 180,E1 -24324.832,E2 -24324.832} C_VEL
LIN {X 0,Y 178.044,Z 432.093,A -85,B 0,C 180,E1 -24328.982,E2 -24328.982} C_VEL
LIN {X 0,Y 180.757,Z 439.219,A -85,B 0,C 180,E1 -24332.979,E2 -24332.979} C_VEL
LIN {X 0,Y 182.604,Z 445.546,A -85,B 0,C 180,E1 -24336.074,E2 -24336.074} C_VEL
LIN {X 0,Y 183.417,Z 451.722,A -85,B 0,C 180,E1 -24338.624,E2 -24338.624} C_VEL
LIN {X 0,Y 183.595,Z 459.969,A -85,B 0,C 180,E1 -24341.751,E2 -24341.751} C_VEL
LIN {X 0,Y 183.149,Z 462.651,A -85,B 0,C 180,E1 -24342.656,E2 -24342.656} C_VEL
LIN {X 0,Y 177.082,Z 473.701,A -85,B 0,C 180,E1 -24345.213,E2 -24345.213} C_VEL
LIN {X 0,Y 171.864,Z 482.607,A -85,B 0,C 180,E1 -24347.835,E2 -24347.835} C_VEL
LIN {X 0,Y 165.715,Z 491.98,A -85,B 0,C 180,E1 -24351.276,E2 -24351.276} C_VEL
LIN {X 0,Y 159.906,Z 500.189,A -85,B 0,C 180,E1 -24355.154,E2 -24355.154} C_VEL
LIN {X 0,Y 154.104,Z 507.892,A -85,B 0,C 180,E1 -24359.889,E2 -24359.889} C_VEL
LIN {X 0,Y 149.442,Z 514.005,A -85,B 0,C 180,E1 -24364.959,E2 -24364.959} C_VEL
LIN {X 0,Y 145.752,Z 518.716,A -85,B 0,C 180,E1 -24370.272,E2 -24370.272} C_VEL
LIN {X 0,Y 143.184,Z 522.154,A -85,B 0,C 180,E1 -24375.792,E2 -24375.792} C_VEL
LIN {X 0,Y 141.659,Z 524.415,A -85,B 0,C 180,E1 -24381.439,E2 -24381.439} C_VEL
LIN {X 0,Y 141.057,Z 525.558,A -85,B 0,C 180,E1 -24387.143,E2 -24387.143} C_VEL
LIN {X 0,Y 141.019,Z 525.709,A -85,B 0,C 180,E1 -24389.999,E2 -24389.999} C_VEL
LIN {X 0,Y 141.262,Z 525.155,A -85,B 0,C 180,E1 -24395.709,E2 -24395.709} C_VEL
LIN {X 0,Y 142.252,Z 523.504,A -85,B 0,C 180,E1 -24401.397,E2 -24401.397} C_VEL
LIN {X 0,Y 144.306,Z 520.701,A -85,B 0,C 180,E1 -24406.989,E2 -24406.989} C_VEL
LIN {X 0,Y 147.34,Z 516.682,A -85,B 0,C 180,E1 -24412.431,E2 -24412.431} C_VEL
LIN {X 0,Y 151.511,Z 511.338,A -85,B 0,C 180,E1 -24417.635,E2 -24417.635} C_VEL
LIN {X 0,Y 156.805,Z 504.51,A -85,B 0,C 180,E1 -24422.535,E2 -24422.535} C_VEL
LIN {X 0,Y 163.066,Z 495.976,A -85,B 0,C 180,E1 -24427.111,E2 -24427.111} C_VEL
LIN {X 0,Y 169.286,Z 486.889,A -85,B 0,C 180,E1 -24430.832,E2 -24430.832} C_VEL
LIN {X 0,Y 174.929,Z 477.641,A -85,B 0,C 180,E1 -24433.87,E2 -24433.87} C_VEL
LIN {X 0,Y 181.229,Z 466.622,A -85,B 0,C 180,E1 -24436.644,E2 -24436.644} C_VEL
LIN {X 0,Y 183.077,Z 463.12,A -85,B 0,C 180,E1 -24437.384,E2 -24437.384} C_VEL
LIN {X 0,Y 183.593,Z 461.686,A -85,B 0,C 180,E1 -24437.764,E2 -24437.764} C_VEL
LIN {X 0,Y 183.651,Z 453.558,A -85,B 0,C 180,E1 -24440.841,E2 -24440.841} C_VEL
LIN {X 0,Y 183.203,Z 448.044,A -85,B 0,C 180,E1 -24443.018,E2 -24443.018} C_VEL
LIN {X 0,Y 181.758,Z 442.123,A -85,B 0,C 180,E1 -24445.764,E2 -24445.764} C_VEL
LIN {X 0,Y 179.248,Z 434.937,A -85,B 0,C 180,E1 -24449.606,E2 -24449.606} C_VEL
LIN {X 0,Y 177.07,Z 429.527,A -85,B 0,C 180,E1 -24452.842,E2 -24452.842} C_VEL
LIN {X 0,Y 173.991,Z 423.29,A -85,B 0,C 180,E1 -24457.435,E2 -24457.435} C_VEL
LIN {X 0,Y 172.961,Z 421.252,A -85,B 0,C 180,E1 -24459.155,E2 -24459.155} C_VEL
LIN {X 0,Y 170.731,Z 417.089,A -85,B 0,C 180,E1 -24463.253,E2 -24463.253} C_VEL
LIN {X 0,Y 169.114,Z 414.469,A -85,B 0,C 180,E1 -24466.787,E2 -24466.787} C_VEL
LIN {X 0,Y 168.806,Z 413.245,A -85,B 0,C 180,E1 -24467.985,E2 -24467.985} C_VEL
LIN {X 0,Y 167.267,Z 411.474,A -85,B 0,C 180,E1 -24472.758,E2 -24472.758} C_VEL
LIN {X 0,Y 166.862,Z 409.648,A -85,B 0,C 180,E1 -24480,E2 -24480} C_VEL
LIN {X 0,Y 167.792,Z 411.924,A -85,B 0,C 180,E1 -24487.218,E2 -24487.218} C_VEL
LIN {X 0,Y 169.009,Z 413.726,A -85,B 0,C 180,E1 -24490.785,E2 -24490.785} C_VEL
LIN {X 0,Y 170.763,Z 418.794,A -85,B 0,C 180,E1 -24495.516,E2 -24495.516} C_VEL
LIN {X 0,Y 171.431,Z 419.899,A -85,B 0,C 180,E1 -24496.677,E2 -24496.677} C_VEL
LIN {X 0,Y 173.873,Z 426.421,A -85,B 0,C 180,E1 -24501.332,E2 -24501.332} C_VEL
LIN {X 0,Y 175.579,Z 431.215,A -85,B 0,C 180,E1 -24504.222,E2 -24504.222} C_VEL
LIN {X 0,Y 177.528,Z 437.476,A -85,B 0,C 180,E1 -24507.479,E2 -24507.479} C_VEL
LIN {X 0,Y 179.685,Z 445.521,A -85,B 0,C 180,E1 -24511.214,E2 -24511.214} C_VEL
LIN {X 0,Y 181.009,Z 452.963,A -85,B 0,C 180,E1 -24514.224,E2 -24514.224} C_VEL
LIN {X 0,Y 180.893,Z 460.45,A -85,B 0,C 180,E1 -24516.667,E2 -24516.667} C_VEL
LIN {X 0,Y 179.858,Z 469.447,A -85,B 0,C 180,E1 -24519.449,E2 -24519.449} C_VEL
LIN {X 0,Y 178.226,Z 477.935,A -85,B 0,C 180,E1 -24522.095,E2 -24522.095} C_VEL
LIN {X 0,Y 177.277,Z 481.411,A -85,B 0,C 180,E1 -24523.21,E2 -24523.21} C_VEL
LIN {X 0,Y 171.414,Z 491.383,A -85,B 0,C 180,E1 -24525.814,E2 -24525.814} C_VEL
LIN {X 0,Y 164.601,Z 501.988,A -85,B 0,C 180,E1 -24529.375,E2 -24529.375} C_VEL
LIN {X 0,Y 158.687,Z 510.839,A -85,B 0,C 180,E1 -24533.282,E2 -24533.282} C_VEL
LIN {X 0,Y 154.184,Z 517.258,A -85,B 0,C 180,E1 -24536.841,E2 -24536.841} C_VEL
LIN {X 0,Y 149.02,Z 524.31,A -85,B 0,C 180,E1 -24541.862,E2 -24541.862} C_VEL
LIN {X 0,Y 145.144,Z 529.879,A -85,B 0,C 180,E1 -24547.211,E2 -24547.211} C_VEL
LIN {X 0,Y 142.469,Z 534.108,A -85,B 0,C 180,E1 -24552.785,E2 -24552.785} C_VEL
LIN {X 0,Y 141,Z 537.093,A -85,B 0,C 180,E1 -24558.501,E2 -24558.501} C_VEL
LIN {X 0,Y 140.637,Z 538.896,A -85,B 0,C 180,E1 -24564.265,E2 -24564.265} C_VEL
LIN {X 0,Y 140.735,Z 539.36,A -85,B 0,C 180,E1 -24567.139,E2 -24567.139} C_VEL
LIN {X 0,Y 140.877,Z 539.526,A -85,B 0,C 180,E1 -24570.001,E2 -24570.001} C_VEL
LIN {X 0,Y 140.735,Z 539.354,A -85,B 0,C 180,E1 -24572.864,E2 -24572.864} C_VEL
LIN {X 0,Y 140.722,Z 538.112,A -85,B 0,C 180,E1 -24578.618,E2 -24578.618} C_VEL
LIN {X 0,Y 141.558,Z 535.7,A -85,B 0,C 180,E1 -24584.374,E2 -24584.374} C_VEL
LIN {X 0,Y 143.664,Z 532.089,A -85,B 0,C 180,E1 -24590.027,E2 -24590.027} C_VEL
LIN {X 0,Y 146.941,Z 527.184,A -85,B 0,C 180,E1 -24595.498,E2 -24595.498} C_VEL
LIN {X 0,Y 151.392,Z 520.859,A -85,B 0,C 180,E1 -24600.708,E2 -24600.708} C_VEL
LIN {X 0,Y 157.101,Z 512.95,A -85,B 0,C 180,E1 -24605.562,E2 -24605.562} C_VEL
LIN {X 0,Y 162.823,Z 504.547,A -85,B 0,C 180,E1 -24609.544,E2 -24609.544} C_VEL
LIN {X 0,Y 169.431,Z 494.452,A -85,B 0,C 180,E1 -24613.191,E2 -24613.191} C_VEL
LIN {X 0,Y 175.634,Z 484.149,A -85,B 0,C 180,E1 -24616.078,E2 -24616.078} C_VEL
LIN {X 0,Y 177.256,Z 481.193,A -85,B 0,C 180,E1 -24616.784,E2 -24616.784} C_VEL
LIN {X 0,Y 178.091,Z 478.062,A -85,B 0,C 180,E1 -24617.792,E2 -24617.792} C_VEL
LIN {X 0,Y 178.483,Z 474.182,A -85,B 0,C 180,E1 -24619.215,E2 -24619.215} C_VEL
LIN {X 0,Y 177.976,Z 470.658,A -85,B 0,C 180,E1 -24620.746,E2 -24620.746} C_VEL
LIN {X 0,Y 175.793,Z 461.477,A -85,B 0,C 180,E1 -24624.96,E2 -24624.96} C_VEL
LIN {X 0,Y 175.775,Z 458.843,A -85,B 0,C 180,E1 -24625.948,E2 -24625.948} C_VEL
LIN {X 0,Y 175.72,Z 455.62,A -85,B 0,C 180,E1 -24627.132,E2 -24627.132} C_VEL
LIN {X 0,Y 174.215,Z 446.845,A -85,B 0,C 180,E1 -24631.047,E2 -24631.047} C_VEL
LIN {X 0,Y 172.493,Z 439.733,A -85,B 0,C 180,E1 -24634.672,E2 -24634.672} C_VEL
LIN {X 0,Y 171.375,Z 435.501,A -85,B 0,C 180,E1 -24637.071,E2 -24637.071} C_VEL
LIN {X 0,Y 169.547,Z 430.197,A -85,B 0,C 180,E1 -24640.634,E2 -24640.634} C_VEL
LIN {X 0,Y 168.117,Z 425.672,A -85,B 0,C 180,E1 -24644.052,E2 -24644.052} C_VEL
LIN {X 0,Y 166.314,Z 420.751,A -85,B 0,C 180,E1 -24649.038,E2 -24649.038} C_VEL
LIN {X 0,Y 165.28,Z 418.518,A -85,B 0,C 180,E1 -24652.671,E2 -24652.671} C_VEL
LIN {X 0,Y 164.454,Z 415.917,A -85,B 0,C 180,E1 -24660,E2 -24660} C_VEL
LIN {X 0,Y 165.325,Z 418.692,A -85,B 0,C 180,E1 -24669.79,E2 -24669.79} C_VEL
LIN {X 0,Y 166.062,Z 419.924,A -85,B 0,C 180,E1 -24672.217,E2 -24672.217} C_VEL
LIN {X 0,Y 168.339,Z 424.944,A -85,B 0,C 180,E1 -24678.248,E2 -24678.248} C_VEL
LIN {X 0,Y 170.193,Z 428.647,A -85,B 0,C 180,E1 -24681.818,E2 -24681.818} C_VEL
LIN {X 0,Y 171.494,Z 431.513,A -85,B 0,C 180,E1 -24684.193,E2 -24684.193} C_VEL
LIN {X 0,Y 173.527,Z 436.627,A -85,B 0,C 180,E1 -24687.76,E2 -24687.76} C_VEL
LIN {X 0,Y 175.924,Z 443.558,A -85,B 0,C 180,E1 -24691.961,E2 -24691.961} C_VEL
LIN {X 0,Y 177.472,Z 449.403,A -85,B 0,C 180,E1 -24695.045,E2 -24695.045} C_VEL
LIN {X 0,Y 178.061,Z 454.069,A -85,B 0,C 180,E1 -24697.146,E2 -24697.146} C_VEL
LIN {X 0,Y 178.024,Z 461.719,A -85,B 0,C 180,E1 -24700.273,E2 -24700.273} C_VEL
LIN {X 0,Y 177.677,Z 464.403,A -85,B 0,C 180,E1 -24701.275,E2 -24701.275} C_VEL
LIN {X 0,Y 171.04,Z 475.819,A -85,B 0,C 180,E1 -24704.021,E2 -24704.021} C_VEL
LIN {X 0,Y 165.791,Z 484.28,A -85,B 0,C 180,E1 -24706.657,E2 -24706.657} C_VEL
LIN {X 0,Y 159.344,Z 493.584,A -85,B 0,C 180,E1 -24710.242,E2 -24710.242} C_VEL
LIN {X 0,Y 153.311,Z 501.619,A -85,B 0,C 180,E1 -24714.233,E2 -24714.233} C_VEL
LIN {X 0,Y 147.09,Z 509.334,A -85,B 0,C 180,E1 -24719.322,E2 -24719.322} C_VEL
LIN {X 0,Y 141.931,Z 515.658,A -85,B 0,C 180,E1 -24725.108,E2 -24725.108} C_VEL
LIN {X 0,Y 139.051,Z 519.067,A -85,B 0,C 180,E1 -24729.279,E2 -24729.279} C_VEL
LIN {X 0,Y 136.306,Z 522.503,A -85,B 0,C 180,E1 -24735.059,E2 -24735.059} C_VEL
LIN {X 0,Y 134.635,Z 524.763,A -85,B 0,C 180,E1 -24740.989,E2 -24740.989} C_VEL
LIN {X 0,Y 133.974,Z 525.905,A -85,B 0,C 180,E1 -24746.992,E2 -24746.992} C_VEL
LIN {X 0,Y 133.928,Z 526.056,A -85,B 0,C 180,E1 -24749.999,E2 -24749.999} C_VEL
LIN {X 0,Y 134.21,Z 525.502,A -85,B 0,C 180,E1 -24756.01,E2 -24756.01} C_VEL
LIN {X 0,Y 135.301,Z 523.851,A -85,B 0,C 180,E1 -24761.991,E2 -24761.991} C_VEL
LIN {X 0,Y 137.512,Z 521.049,A -85,B 0,C 180,E1 -24767.856,E2 -24767.856} C_VEL
LIN {X 0,Y 140.796,Z 517.03,A -85,B 0,C 180,E1 -24773.535,E2 -24773.535} C_VEL
LIN {X 0,Y 145.232,Z 511.686,A -85,B 0,C 180,E1 -24778.94,E2 -24778.94} C_VEL
LIN {X 0,Y 150.854,Z 504.858,A -85,B 0,C 180,E1 -24783.989,E2 -24783.989} C_VEL
LIN {X 0,Y 157.463,Z 496.322,A -85,B 0,C 180,E1 -24788.67,E2 -24788.67} C_VEL
LIN {X 0,Y 162.987,Z 488.643,A -85,B 0,C 180,E1 -24791.939,E2 -24791.939} C_VEL
LIN {X 0,Y 169.88,Z 477.986,A -85,B 0,C 180,E1 -24795.53,E2 -24795.53} C_VEL
LIN {X 0,Y 176.433,Z 466.967,A -85,B 0,C 180,E1 -24798.32,E2 -24798.32} C_VEL
LIN {X 0,Y 177.583,Z 464.915,A -85,B 0,C 180,E1 -24798.757,E2 -24798.757} C_VEL
LIN {X 0,Y 178.009,Z 463.514,A -85,B 0,C 180,E1 -24799.178,E2 -24799.178} C_VEL
LIN {X 0,Y 178.216,Z 456.36,A -85,B 0,C 180,E1 -24802.063,E2 -24802.063} C_VEL
LIN {X 0,Y 177.867,Z 451.023,A -85,B 0,C 180,E1 -24804.351,E2 -24804.351} C_VEL
LIN {X 0,Y 176.396,Z 445.009,A -85,B 0,C 180,E1 -24807.46,E2 -24807.46} C_VEL
LIN {X 0,Y 174.404,Z 438.776,A -85,B 0,C 180,E1 -24811.081,E2 -24811.081} C_VEL
LIN {X 0,Y 173.088,Z 435.092,A -85,B 0,C 180,E1 -24813.471,E2 -24813.471} C_VEL
LIN {X 0,Y 170.404,Z 428.978,A -85,B 0,C 180,E1 -24818.211,E2 -24818.211} C_VEL
LIN {X 0,Y 168.087,Z 424.01,A -85,B 0,C 180,E1 -24822.981,E2 -24822.981} C_VEL
LIN {X 0,Y 166.248,Z 420.332,A -85,B 0,C 180,E1 -24827.797,E2 -24827.797} C_VEL
LIN {X 0,Y 165.561,Z 418.957,A -85,B 0,C 180,E1 -24830.224,E2 -24830.224} C_VEL
LIN {X 0,Y 164.607,Z 416.407,A -85,B 0,C 180,E1 -24840,E2 -24840} C_VEL
LIN {X 0,Y 165.504,Z 418.733,A -85,B 0,C 180,E1 -24847.319,E2 -24847.319} C_VEL
LIN {X 0,Y 166.23,Z 419.91,A -85,B 0,C 180,E1 -24849.736,E2 -24849.736} C_VEL
LIN {X 0,Y 168.46,Z 426.483,A -85,B 0,C 180,E1 -24856.358,E2 -24856.358} C_VEL
LIN {X 0,Y 170.301,Z 432.071,A -85,B 0,C 180,E1 -24860.535,E2 -24860.535} C_VEL
LIN {X 0,Y 171.768,Z 436.809,A -85,B 0,C 180,E1 -24863.511,E2 -24863.511} C_VEL
LIN {X 0,Y 173.737,Z 444.36,A -85,B 0,C 180,E1 -24867.592,E2 -24867.592} C_VEL
LIN {X 0,Y 175.18,Z 451.351,A -85,B 0,C 180,E1 -24870.905,E2 -24870.905} C_VEL
LIN {X 0,Y 175.925,Z 457.025,A -85,B 0,C 180,E1 -24873.318,E2 -24873.318} C_VEL
LIN {X 0,Y 175.405,Z 464.635,A -85,B 0,C 180,E1 -24875.909,E2 -24875.909} C_VEL
LIN {X 0,Y 173.781,Z 474.286,A -85,B 0,C 180,E1 -24879.097,E2 -24879.097} C_VEL
LIN {X 0,Y 171.883,Z 481.741,A -85,B 0,C 180,E1 -24881.571,E2 -24881.571} C_VEL
LIN {X 0,Y 170.743,Z 484.036,A -85,B 0,C 180,E1 -24882.193,E2 -24882.193} C_VEL
LIN {X 0,Y 164.269,Z 494.315,A -85,B 0,C 180,E1 -24885.097,E2 -24885.097} C_VEL
LIN {X 0,Y 157.339,Z 504.372,A -85,B 0,C 180,E1 -24888.789,E2 -24888.789} C_VEL
LIN {X 0,Y 150.486,Z 513.836,A -85,B 0,C 180,E1 -24893.457,E2 -24893.457} C_VEL
LIN {X 0,Y 145.271,Z 520.628,A -85,B 0,C 180,E1 -24897.85,E2 -24897.85} C_VEL
LIN {X 0,Y 140.472,Z 526.918,A -85,B 0,C 180,E1 -24903.24,E2 -24903.24} C_VEL
LIN {X 0,Y 136.938,Z 531.803,A -85,B 0,C 180,E1 -24908.947,E2 -24908.947} C_VEL
LIN {X 0,Y 134.615,Z 535.399,A -85,B 0,C 180,E1 -24914.87,E2 -24914.87} C_VEL
LIN {X 0,Y 133.651,Z 537.791,A -85,B 0,C 180,E1 -24920.925,E2 -24920.925} C_VEL
LIN {X 0,Y 133.634,Z 539.012,A -85,B 0,C 180,E1 -24926.987,E2 -24926.987} C_VEL
LIN {X 0,Y 133.786,Z 539.178,A -85,B 0,C 180,E1 -24930.001,E2 -24930.001} C_VEL
LIN {X 0,Y 133.635,Z 539.006,A -85,B 0,C 180,E1 -24933.016,E2 -24933.016} C_VEL
LIN {X 0,Y 133.663,Z 537.762,A -85,B 0,C 180,E1 -24939.077,E2 -24939.077} C_VEL
LIN {X 0,Y 134.619,Z 535.348,A -85,B 0,C 180,E1 -24945.133,E2 -24945.133} C_VEL
LIN {X 0,Y 136.946,Z 531.736,A -85,B 0,C 180,E1 -24951.055,E2 -24951.055} C_VEL
LIN {X 0,Y 140.474,Z 526.83,A -85,B 0,C 180,E1 -24956.763,E2 -24956.763} C_VEL
LIN {X 0,Y 145.267,Z 520.506,A -85,B 0,C 180,E1 -24962.154,E2 -24962.154} C_VEL
LIN {X 0,Y 151.331,Z 512.597,A -85,B 0,C 180,E1 -24967.139,E2 -24967.139} C_VEL
LIN {X 0,Y 157.356,Z 504.193,A -85,B 0,C 180,E1 -24971.208,E2 -24971.208} C_VEL
LIN {X 0,Y 164.28,Z 494.099,A -85,B 0,C 180,E1 -24974.902,E2 -24974.902} C_VEL
LIN {X 0,Y 170.757,Z 483.796,A -85,B 0,C 180,E1 -24977.805,E2 -24977.805} C_VEL
LIN {X 0,Y 171.849,Z 481.498,A -85,B 0,C 180,E1 -24978.434,E2 -24978.434} C_VEL
LIN {X 0,Y 174.046,Z 472.402,A -85,B 0,C 180,E1 -24981.463,E2 -24981.463} C_VEL
LIN {X 0,Y 175.42,Z 463.177,A -85,B 0,C 180,E1 -24984.495,E2 -24984.495} C_VEL
LIN {X 0,Y 175.775,Z 458.843,A -85,B 0,C 180,E1 -24985.948,E2 -24985.948} C_VEL
LIN {X 0,Y 175.618,Z 456.406,A -85,B 0,C 180,E1 -24986.939,E2 -24986.939} C_VEL
LIN {X 0,Y 174.434,Z 453.563,A -85,B 0,C 180,E1 -24988.586,E2 -24988.586} C_VEL
LIN {X 0,Y 171.316,Z 450.099,A -85,B 0,C 180,E1 -24991.546,E2 -24991.546} C_VEL
LIN {X 0,Y 169.047,Z 447.232,A -85,B 0,C 180,E1 -24994.014,E2 -24994.014} C_VEL
LIN {X 0,Y 168.379,Z 445.368,A -85,B 0,C 180,E1 -24995.225,E2 -24995.225} C_VEL
LIN {X 0,Y 167.429,Z 440.996,A -85,B 0,C 180,E1 -24997.804,E2 -24997.804} C_VEL
LIN {X 0,Y 165.945,Z 435.79,A -85,B 0,C 180,E1 -25001.48,E2 -25001.48} C_VEL
LIN {X 0,Y 164.644,Z 431.306,A -85,B 0,C 180,E1 -25005.161,E2 -25005.161} C_VEL
LIN {X 0,Y 163.321,Z 426.689,A -85,B 0,C 180,E1 -25010.089,E2 -25010.089} C_VEL
LIN {X 0,Y 162.696,Z 425.246,A -85,B 0,C 180,E1 -25012.554,E2 -25012.554} C_VEL
LIN {X 0,Y 161.946,Z 422.593,A -85,B 0,C 180,E1 -25020,E2 -25020} C_VEL
LIN {X 0,Y 162.668,Z 425.389,A -85,B 0,C 180,E1 -25029.952,E2 -25029.952} C_VEL
LIN {X 0,Y 163.263,Z 426.809,A -85,B 0,C 180,E1 -25032.43,E2 -25032.43} C_VEL
LIN {X 0,Y 165.33,Z 431.844,A -85,B 0,C 180,E1 -25038.592,E2 -25038.592} C_VEL
LIN {X 0,Y 166.99,Z 435.65,A -85,B 0,C 180,E1 -25042.258,E2 -25042.258} C_VEL
LIN {X 0,Y 169.314,Z 442.063,A -85,B 0,C 180,E1 -25047.168,E2 -25047.168} C_VEL
LIN {X 0,Y 171.366,Z 448.873,A -85,B 0,C 180,E1 -25051.527,E2 -25051.527} C_VEL
LIN {X 0,Y 172.557,Z 454.769,A -85,B 0,C 180,E1 -25054.765,E2 -25054.765} C_VEL
LIN {X 0,Y 172.737,Z 459.299,A -85,B 0,C 180,E1 -25056.878,E2 -25056.878} C_VEL
LIN {X 0,Y 172.362,Z 465.826,A -85,B 0,C 180,E1 -25059.678,E2 -25059.678} C_VEL
LIN {X 0,Y 167.306,Z 474.403,A -85,B 0,C 180,E1 -25061.786,E2 -25061.786} C_VEL
LIN {X 0,Y 161.31,Z 483.716,A -85,B 0,C 180,E1 -25064.584,E2 -25064.584} C_VEL
LIN {X 0,Y 154.875,Z 492.681,A -85,B 0,C 180,E1 -25067.983,E2 -25067.983} C_VEL
LIN {X 0,Y 148.449,Z 500.89,A -85,B 0,C 180,E1 -25072.014,E2 -25072.014} C_VEL
LIN {X 0,Y 141.982,Z 508.592,A -85,B 0,C 180,E1 -25077.009,E2 -25077.009} C_VEL
LIN {X 0,Y 136.669,Z 514.705,A -85,B 0,C 180,E1 -25082.43,E2 -25082.43} C_VEL
LIN {X 0,Y 132.399,Z 519.418,A -85,B 0,C 180,E1 -25088.186,E2 -25088.186} C_VEL
LIN {X 0,Y 129.463,Z 522.851,A -85,B 0,C 180,E1 -25094.249,E2 -25094.249} C_VEL
LIN {X 0,Y 127.62,Z 525.112,A -85,B 0,C 180,E1 -25100.489,E2 -25100.489} C_VEL
LIN {X 0,Y 126.887,Z 526.253,A -85,B 0,C 180,E1 -25106.824,E2 -25106.824} C_VEL
LIN {X 0,Y 126.839,Z 526.404,A -85,B 0,C 180,E1 -25109.999,E2 -25109.999} C_VEL
LIN {X 0,Y 127.164,Z 525.849,A -85,B 0,C 180,E1 -25116.345,E2 -25116.345} C_VEL
LIN {X 0,Y 128.355,Z 524.199,A -85,B 0,C 180,E1 -25122.65,E2 -25122.65} C_VEL
LIN {X 0,Y 130.739,Z 521.398,A -85,B 0,C 180,E1 -25128.815,E2 -25128.815} C_VEL
LIN {X 0,Y 134.313,Z 517.377,A -85,B 0,C 180,E1 -25134.745,E2 -25134.745} C_VEL
LIN {X 0,Y 139.041,Z 512.034,A -85,B 0,C 180,E1 -25140.361,E2 -25140.361} C_VEL
LIN {X 0,Y 144.998,Z 505.205,A -85,B 0,C 180,E1 -25145.564,E2 -25145.564} C_VEL
LIN {X 0,Y 151.975,Z 496.668,A -85,B 0,C 180,E1 -25150.346,E2 -25150.346} C_VEL
LIN {X 0,Y 157.783,Z 488.988,A -85,B 0,C 180,E1 -25153.66,E2 -25153.66} C_VEL
LIN {X 0,Y 164.986,Z 478.331,A -85,B 0,C 180,E1 -25157.289,E2 -25157.289} C_VEL
LIN {X 0,Y 171.8,Z 467.311,A -85,B 0,C 180,E1 -25160.086,E2 -25160.086} C_VEL
LIN {X 0,Y 172.401,Z 466.319,A -85,B 0,C 180,E1 -25160.303,E2 -25160.303} C_VEL
LIN {X 0,Y 172.842,Z 459.652,A -85,B 0,C 180,E1 -25163.148,E2 -25163.148} C_VEL
LIN {X 0,Y 172.62,Z 454.395,A -85,B 0,C 180,E1 -25165.606,E2 -25165.606} C_VEL
LIN {X 0,Y 171.213,Z 448.181,A -85,B 0,C 180,E1 -25169.13,E2 -25169.13} C_VEL
LIN {X 0,Y 169.505,Z 442.363,A -85,B 0,C 180,E1 -25172.865,E2 -25172.865} C_VEL
LIN {X 0,Y 167.688,Z 437.27,A -85,B 0,C 180,E1 -25176.668,E2 -25176.668} C_VEL
LIN {X 0,Y 166.088,Z 433.26,A -85,B 0,C 180,E1 -25180.213,E2 -25180.213} C_VEL
LIN {X 0,Y 165.105,Z 430.939,A -85,B 0,C 180,E1 -25182.664,E2 -25182.664} C_VEL
LIN {X 0,Y 163.456,Z 427.158,A -85,B 0,C 180,E1 -25187.585,E2 -25187.585} C_VEL
LIN {X 0,Y 162.877,Z 425.69,A -85,B 0,C 180,E1 -25190.061,E2 -25190.061} C_VEL
LIN {X 0,Y 161.867,Z 423.678,A -85,B 0,C 180,E1 -25197.511,E2 -25197.511} C_VEL
LIN {X 0,Y 162.081,Z 423.074,A -85,B 0,C 180,E1 -25200,E2 -25200} C_VEL
LIN {X 0,Y 162.92,Z 425.45,A -85,B 0,C 180,E1 -25207.435,E2 -25207.435} C_VEL
LIN {X 0,Y 163.557,Z 426.832,A -85,B 0,C 180,E1 -25209.897,E2 -25209.897} C_VEL
LIN {X 0,Y 165.103,Z 432.381,A -85,B 0,C 180,E1 -25215.604,E2 -25215.604} C_VEL
LIN {X 0,Y 166.585,Z 437.62,A -85,B 0,C 180,E1 -25219.725,E2 -25219.725} C_VEL
LIN {X 0,Y 167.822,Z 442.464,A -85,B 0,C 180,E1 -25222.885,E2 -25222.885} C_VEL
LIN {X 0,Y 169.411,Z 450.016,A -85,B 0,C 180,E1 -25227.15,E2 -25227.15} C_VEL
LIN {X 0,Y 170.548,Z 457.876,A -85,B 0,C 180,E1 -25231.003,E2 -25231.003} C_VEL
LIN {X 0,Y 170.742,Z 460.9,A -85,B 0,C 180,E1 -25232.35,E2 -25232.35} C_VEL
LIN {X 0,Y 169.928,Z 467.824,A -85,B 0,C 180,E1 -25234.836,E2 -25234.836} C_VEL
LIN {X 0,Y 168.371,Z 475.575,A -85,B 0,C 180,E1 -25237.527,E2 -25237.527} C_VEL
LIN {X 0,Y 166.02,Z 483.688,A -85,B 0,C 180,E1 -25240.363,E2 -25240.363} C_VEL
LIN {X 0,Y 159.286,Z 493.967,A -85,B 0,C 180,E1 -25243.282,E2 -25243.282} C_VEL
LIN {X 0,Y 152.015,Z 504.023,A -85,B 0,C 180,E1 -25247.007,E2 -25247.007} C_VEL
LIN {X 0,Y 145.655,Z 512.4,A -85,B 0,C 180,E1 -25251.153,E2 -25251.153} C_VEL
LIN {X 0,Y 140.787,Z 518.444,A -85,B 0,C 180,E1 -25254.967,E2 -25254.967} C_VEL
LIN {X 0,Y 135.241,Z 525.114,A -85,B 0,C 180,E1 -25260.419,E2 -25260.419} C_VEL
LIN {X 0,Y 131.064,Z 530.389,A -85,B 0,C 180,E1 -25266.335,E2 -25266.335} C_VEL
LIN {X 0,Y 128.839,Z 533.407,A -85,B 0,C 180,E1 -25270.897,E2 -25270.897} C_VEL
LIN {X 0,Y 126.975,Z 536.391,A -85,B 0,C 180,E1 -25277.21,E2 -25277.21} C_VEL
LIN {X 0,Y 126.448,Z 538.197,A -85,B 0,C 180,E1 -25283.619,E2 -25283.619} C_VEL
LIN {X 0,Y 126.576,Z 538.733,A -85,B 0,C 180,E1 -25288.052,E2 -25288.052} C_VEL
LIN {X 0,Y 126.687,Z 538.831,A -85,B 0,C 180,E1 -25290.001,E2 -25290.001} C_VEL
LIN {X 0,Y 126.545,Z 538.658,A -85,B 0,C 180,E1 -25293.185,E2 -25293.185} C_VEL
LIN {X 0,Y 126.6,Z 537.411,A -85,B 0,C 180,E1 -25299.588,E2 -25299.588} C_VEL
LIN {X 0,Y 127.707,Z 534.996,A -85,B 0,C 180,E1 -25305.973,E2 -25305.973} C_VEL
LIN {X 0,Y 130.276,Z 531.384,A -85,B 0,C 180,E1 -25312.188,E2 -25312.188} C_VEL
LIN {X 0,Y 134.092,Z 526.476,A -85,B 0,C 180,E1 -25318.147,E2 -25318.147} C_VEL
LIN {X 0,Y 139.241,Z 520.152,A -85,B 0,C 180,E1 -25323.727,E2 -25323.727} C_VEL
LIN {X 0,Y 145.675,Z 512.243,A -85,B 0,C 180,E1 -25328.844,E2 -25328.844} C_VEL
LIN {X 0,Y 152.028,Z 503.839,A -85,B 0,C 180,E1 -25332.991,E2 -25332.991} C_VEL
LIN {X 0,Y 159.291,Z 493.745,A -85,B 0,C 180,E1 -25336.719,E2 -25336.719} C_VEL
LIN {X 0,Y 166.015,Z 483.441,A -85,B 0,C 180,E1 -25339.643,E2 -25339.643} C_VEL
LIN {X 0,Y 168.669,Z 473.668,A -85,B 0,C 180,E1 -25343.06,E2 -25343.06} C_VEL
LIN {X 0,Y 170.085,Z 465.989,A -85,B 0,C 180,E1 -25345.733,E2 -25345.733} C_VEL
LIN {X 0,Y 170.636,Z 460.723,A -85,B 0,C 180,E1 -25347.627,E2 -25347.627} C_VEL
LIN {X 0,Y 169.887,Z 453.563,A -85,B 0,C 180,E1 -25350.917,E2 -25350.917} C_VEL
LIN {X 0,Y 168.581,Z 446.282,A -85,B 0,C 180,E1 -25354.703,E2 -25354.703} C_VEL
LIN {X 0,Y 168.379,Z 445.368,A -85,B 0,C 180,E1 -25355.225,E2 -25355.225} C_VEL
LIN {X 0,Y 167.351,Z 442.953,A -85,B 0,C 180,E1 -25357.026,E2 -25357.026} C_VEL
LIN {X 0,Y 165.813,Z 441.453,A -85,B 0,C 180,E1 -25358.932,E2 -25358.932} C_VEL
LIN {X 0,Y 161.759,Z 438.643,A -85,B 0,C 180,E1 -25364.291,E2 -25364.291} C_VEL
LIN {X 0,Y 161.233,Z 437.475,A -85,B 0,C 180,E1 -25365.643,E2 -25365.643} C_VEL
LIN {X 0,Y 160.341,Z 433.525,A -85,B 0,C 180,E1 -25369.903,E2 -25369.903} C_VEL
LIN {X 0,Y 159.826,Z 431.891,A -85,B 0,C 180,E1 -25372.42,E2 -25372.42} C_VEL
LIN {X 0,Y 159.164,Z 429.178,A -85,B 0,C 180,E1 -25380,E2 -25380} C_VEL
LIN {X 0,Y 159.244,Z 431.105,A -85,B 0,C 180,E1 -25387.609,E2 -25387.609} C_VEL
LIN {X 0,Y 159.715,Z 432.027,A -85,B 0,C 180,E1 -25390.138,E2 -25390.138} C_VEL
LIN {X 0,Y 160.206,Z 433.52,A -85,B 0,C 180,E1 -25392.671,E2 -25392.671} C_VEL
LIN {X 0,Y 161.633,Z 437.464,A -85,B 0,C 180,E1 -25397.72,E2 -25397.72} C_VEL
LIN {X 0,Y 163.14,Z 441.533,A -85,B 0,C 180,E1 -25401.884,E2 -25401.884} C_VEL
LIN {X 0,Y 164.887,Z 447.235,A -85,B 0,C 180,E1 -25406.478,E2 -25406.478} C_VEL
LIN {X 0,Y 166.146,Z 452.019,A -85,B 0,C 180,E1 -25409.804,E2 -25409.804} C_VEL
LIN {X 0,Y 167.192,Z 457.443,A -85,B 0,C 180,E1 -25413.125,E2 -25413.125} C_VEL
LIN {X 0,Y 167.43,Z 461.539,A -85,B 0,C 180,E1 -25415.252,E2 -25415.252} C_VEL
LIN {X 0,Y 166.96,Z 467.238,A -85,B 0,C 180,E1 -25417.882,E2 -25417.882} C_VEL
LIN {X 0,Y 166.238,Z 469.136,A -85,B 0,C 180,E1 -25418.544,E2 -25418.544} C_VEL
LIN {X 0,Y 159.189,Z 479.905,A -85,B 0,C 180,E1 -25421.362,E2 -25421.362} C_VEL
LIN {X 0,Y 152.802,Z 489.013,A -85,B 0,C 180,E1 -25424.526,E2 -25424.526} C_VEL
LIN {X 0,Y 145.733,Z 497.927,A -85,B 0,C 180,E1 -25428.462,E2 -25428.462} C_VEL
LIN {X 0,Y 139.347,Z 505.304,A -85,B 0,C 180,E1 -25432.754,E2 -25432.754} C_VEL
LIN {X 0,Y 133.03,Z 512.188,A -85,B 0,C 180,E1 -25438.108,E2 -25438.108} C_VEL
LIN {X 0,Y 127.947,Z 517.578,A -85,B 0,C 180,E1 -25443.931,E2 -25443.931} C_VEL
LIN {X 0,Y 124.078,Z 521.635,A -85,B 0,C 180,E1 -25450.131,E2 -25450.131} C_VEL
LIN {X 0,Y 121.435,Z 524.475,A -85,B 0,C 180,E1 -25456.613,E2 -25456.613} C_VEL
LIN {X 0,Y 120.109,Z 526.167,A -85,B 0,C 180,E1 -25463.278,E2 -25463.278} C_VEL
LIN {X 0,Y 119.753,Z 526.751,A -85,B 0,C 180,E1 -25469.999,E2 -25469.999} C_VEL
LIN {X 0,Y 120.108,Z 526.197,A -85,B 0,C 180,E1 -25476.719,E2 -25476.719} C_VEL
LIN {X 0,Y 121.421,Z 524.548,A -85,B 0,C 180,E1 -25483.385,E2 -25483.385} C_VEL
LIN {X 0,Y 124.009,Z 521.747,A -85,B 0,C 180,E1 -25489.878,E2 -25489.878} C_VEL
LIN {X 0,Y 127.899,Z 517.724,A -85,B 0,C 180,E1 -25496.077,E2 -25496.077} C_VEL
LIN {X 0,Y 132.943,Z 512.382,A -85,B 0,C 180,E1 -25501.913,E2 -25501.913} C_VEL
LIN {X 0,Y 139.277,Z 505.552,A -85,B 0,C 180,E1 -25507.265,E2 -25507.265} C_VEL
LIN {X 0,Y 146.613,Z 497.016,A -85,B 0,C 180,E1 -25512.15,E2 -25512.15} C_VEL
LIN {X 0,Y 152.729,Z 489.333,A -85,B 0,C 180,E1 -25515.498,E2 -25515.498} C_VEL
LIN {X 0,Y 159.12,Z 480.29,A -85,B 0,C 180,E1 -25518.663,E2 -25518.663} C_VEL
LIN {X 0,Y 166.12,Z 469.595,A -85,B 0,C 180,E1 -25521.504,E2 -25521.504} C_VEL
LIN {X 0,Y 167.042,Z 467.679,A -85,B 0,C 180,E1 -25522.078,E2 -25522.078} C_VEL
LIN {X 0,Y 167.555,Z 460.348,A -85,B 0,C 180,E1 -25525.511,E2 -25525.511} C_VEL
LIN {X 0,Y 166.963,Z 455.511,A -85,B 0,C 180,E1 -25528.252,E2 -25528.252} C_VEL
LIN {X 0,Y 165.614,Z 449.465,A -85,B 0,C 180,E1 -25532.173,E2 -25532.173} C_VEL
LIN {X 0,Y 164.651,Z 445.885,A -85,B 0,C 180,E1 -25534.732,E2 -25534.732} C_VEL
LIN {X 0,Y 163.182,Z 441.409,A -85,B 0,C 180,E1 -25538.525,E2 -25538.525} C_VEL
LIN {X 0,Y 161.636,Z 437.039,A -85,B 0,C 180,E1 -25543.048,E2 -25543.048} C_VEL
LIN {X 0,Y 160.386,Z 433.859,A -85,B 0,C 180,E1 -25547.344,E2 -25547.344} C_VEL
LIN {X 0,Y 159.907,Z 432.334,A -85,B 0,C 180,E1 -25549.874,E2 -25549.874} C_VEL
LIN {X 0,Y 159.114,Z 430.757,A -85,B 0,C 180,E1 -25554.932,E2 -25554.932} C_VEL
LIN {X 0,Y 159.29,Z 429.627,A -85,B 0,C 180,E1 -25560,E2 -25560} C_VEL
LIN {X 0,Y 160.052,Z 432.074,A -85,B 0,C 180,E1 -25567.569,E2 -25567.569} C_VEL
LIN {X 0,Y 160.532,Z 433.761,A -85,B 0,C 180,E1 -25570.085,E2 -25570.085} C_VEL
LIN {X 0,Y 161.642,Z 438.481,A -85,B 0,C 180,E1 -25575.122,E2 -25575.122} C_VEL
LIN {X 0,Y 162.718,Z 443.076,A -85,B 0,C 180,E1 -25578.899,E2 -25578.899} C_VEL
LIN {X 0,Y 163.628,Z 447.663,A -85,B 0,C 180,E1 -25582.075,E2 -25582.075} C_VEL
LIN {X 0,Y 164.771,Z 454.959,A -85,B 0,C 180,E1 -25586.402,E2 -25586.402} C_VEL
LIN {X 0,Y 165.469,Z 461.797,A -85,B 0,C 180,E1 -25589.97,E2 -25589.97} C_VEL
LIN {X 0,Y 165.401,Z 465.901,A -85,B 0,C 180,E1 -25591.811,E2 -25591.811} C_VEL
LIN {X 0,Y 163.925,Z 473.566,A -85,B 0,C 180,E1 -25594.676,E2 -25594.676} C_VEL
LIN {X 0,Y 161.552,Z 481.834,A -85,B 0,C 180,E1 -25597.692,E2 -25597.692} C_VEL
LIN {X 0,Y 160.278,Z 485.135,A -85,B 0,C 180,E1 -25598.895,E2 -25598.895} C_VEL
LIN {X 0,Y 153.33,Z 495.136,A -85,B 0,C 180,E1 -25601.857,E2 -25601.857} C_VEL
LIN {X 0,Y 145.829,Z 504.936,A -85,B 0,C 180,E1 -25605.671,E2 -25605.671} C_VEL
LIN {X 0,Y 139.22,Z 513.136,A -85,B 0,C 180,E1 -25609.938,E2 -25609.938} C_VEL
LIN {X 0,Y 133.334,Z 519.927,A -85,B 0,C 180,E1 -25614.565,E2 -25614.565} C_VEL
LIN {X 0,Y 127.798,Z 526.216,A -85,B 0,C 180,E1 -25620.336,E2 -25620.336} C_VEL
LIN {X 0,Y 123.656,Z 531.102,A -85,B 0,C 180,E1 -25626.558,E2 -25626.558} C_VEL
LIN {X 0,Y 120.822,Z 534.697,A -85,B 0,C 180,E1 -25633.093,E2 -25633.093} C_VEL
LIN {X 0,Y 119.552,Z 537.091,A -85,B 0,C 180,E1 -25639.844,E2 -25639.844} C_VEL
LIN {X 0,Y 119.439,Z 538.315,A -85,B 0,C 180,E1 -25646.628,E2 -25646.628} C_VEL
LIN {X 0,Y 119.604,Z 538.483,A -85,B 0,C 180,E1 -25650.001,E2 -25650.001} C_VEL
LIN {X 0,Y 119.44,Z 538.309,A -85,B 0,C 180,E1 -25653.375,E2 -25653.375} C_VEL
LIN {X 0,Y 119.563,Z 537.06,A -85,B 0,C 180,E1 -25660.158,E2 -25660.158} C_VEL
LIN {X 0,Y 120.827,Z 534.644,A -85,B 0,C 180,E1 -25666.909,E2 -25666.909} C_VEL
LIN {X 0,Y 123.663,Z 531.031,A -85,B 0,C 180,E1 -25673.444,E2 -25673.444} C_VEL
LIN {X 0,Y 127.798,Z 526.123,A -85,B 0,C 180,E1 -25679.667,E2 -25679.667} C_VEL
LIN {X 0,Y 133.329,Z 519.799,A -85,B 0,C 180,E1 -25685.44,E2 -25685.44} C_VEL
LIN {X 0,Y 140.154,Z 511.89,A -85,B 0,C 180,E1 -25690.685,E2 -25690.685} C_VEL
LIN {X 0,Y 146.851,Z 503.485,A -85,B 0,C 180,E1 -25694.904,E2 -25694.904} C_VEL
LIN {X 0,Y 154.461,Z 493.391,A -85,B 0,C 180,E1 -25698.657,E2 -25698.657} C_VEL
LIN {X 0,Y 160.289,Z 484.884,A -85,B 0,C 180,E1 -25701.103,E2 -25701.103} C_VEL
LIN {X 0,Y 162.929,Z 476.96,A -85,B 0,C 180,E1 -25704.022,E2 -25704.022} C_VEL
LIN {X 0,Y 164.885,Z 468.158,A -85,B 0,C 180,E1 -25707.262,E2 -25707.262} C_VEL
LIN {X 0,Y 165.431,Z 464.573,A -85,B 0,C 180,E1 -25708.64,E2 -25708.64} C_VEL
LIN {X 0,Y 165.012,Z 457.577,A -85,B 0,C 180,E1 -25712.063,E2 -25712.063} C_VEL
LIN {X 0,Y 164.03,Z 450.49,A -85,B 0,C 180,E1 -25716.02,E2 -25716.02} C_VEL
LIN {X 0,Y 163.322,Z 446.407,A -85,B 0,C 180,E1 -25718.545,E2 -25718.545} C_VEL
LIN {X 0,Y 162.171,Z 441.287,A -85,B 0,C 180,E1 -25722.341,E2 -25722.341} C_VEL
LIN {X 0,Y 161.233,Z 437.475,A -85,B 0,C 180,E1 -25725.643,E2 -25725.643} C_VEL
LIN {X 0,Y 160.406,Z 436.169,A -85,B 0,C 180,E1 -25727.67,E2 -25727.67} C_VEL
LIN {X 0,Y 159.207,Z 435.944,A -85,B 0,C 180,E1 -25729.758,E2 -25729.758} C_VEL
LIN {X 0,Y 156.289,Z 436.868,A -85,B 0,C 180,E1 -25735.52,E2 -25735.52} C_VEL
LIN {X 0,Y 156.045,Z 436.628,A -85,B 0,C 180,E1 -25736.997,E2 -25736.997} C_VEL
LIN {X 0,Y 156.119,Z 435.642,A -85,B 0,C 180,E1 -25740,E2 -25740} C_VEL
LIN {X 0,Y 156.098,Z 437.589,A -85,B 0,C 180,E1 -25747.894,E2 -25747.894} C_VEL
LIN {X 0,Y 156.49,Z 438.548,A -85,B 0,C 180,E1 -25750.349,E2 -25750.349} C_VEL
LIN {X 0,Y 157.415,Z 441.961,A -85,B 0,C 180,E1 -25755.538,E2 -25755.538} C_VEL
LIN {X 0,Y 158.49,Z 445.219,A -85,B 0,C 180,E1 -25759.425,E2 -25759.425} C_VEL
LIN {X 0,Y 159.634,Z 449.405,A -85,B 0,C 180,E1 -25763.343,E2 -25763.343} C_VEL
LIN {X 0,Y 161.014,Z 455.18,A -85,B 0,C 180,E1 -25767.928,E2 -25767.928} C_VEL
LIN {X 0,Y 162.024,Z 461.43,A -85,B 0,C 180,E1 -25772.119,E2 -25772.119} C_VEL
LIN {X 0,Y 162.022,Z 465.663,A -85,B 0,C 180,E1 -25774.495,E2 -25774.495} C_VEL
LIN {X 0,Y 161.496,Z 469.82,A -85,B 0,C 180,E1 -25776.551,E2 -25776.551} C_VEL
LIN {X 0,Y 159.416,Z 473.336,A -85,B 0,C 180,E1 -25777.48,E2 -25777.48} C_VEL
LIN {X 0,Y 152.209,Z 483.624,A -85,B 0,C 180,E1 -25780.463,E2 -25780.463} C_VEL
LIN {X 0,Y 144.614,Z 493.383,A -85,B 0,C 180,E1 -25784.206,E2 -25784.206} C_VEL
LIN {X 0,Y 137.503,Z 501.592,A -85,B 0,C 180,E1 -25788.358,E2 -25788.358} C_VEL
LIN {X 0,Y 130.256,Z 509.294,A -85,B 0,C 180,E1 -25793.592,E2 -25793.592} C_VEL
LIN {X 0,Y 124.225,Z 515.405,A -85,B 0,C 180,E1 -25799.39,E2 -25799.39} C_VEL
LIN {X 0,Y 119.278,Z 520.118,A -85,B 0,C 180,E1 -25805.64,E2 -25805.64} C_VEL
LIN {X 0,Y 115.823,Z 523.55,A -85,B 0,C 180,E1 -25812.337,E2 -25812.337} C_VEL
LIN {X 0,Y 113.635,Z 525.809,A -85,B 0,C 180,E1 -25819.306,E2 -25819.306} C_VEL
LIN {X 0,Y 112.757,Z 526.947,A -85,B 0,C 180,E1 -25826.425,E2 -25826.425} C_VEL
LIN {X 0,Y 112.756,Z 526.957,A -85,B 0,C 180,E1 -25833.572,E2 -25833.572} C_VEL
LIN {X 0,Y 113.632,Z 525.86,A -85,B 0,C 180,E1 -25840.691,E2 -25840.691} C_VEL
LIN {X 0,Y 115.769,Z 523.643,A -85,B 0,C 180,E1 -25847.668,E2 -25847.668} C_VEL
LIN {X 0,Y 119.221,Z 520.245,A -85,B 0,C 180,E1 -25854.369,E2 -25854.369} C_VEL
LIN {X 0,Y 124.154,Z 515.571,A -85,B 0,C 180,E1 -25860.627,E2 -25860.627} C_VEL
LIN {X 0,Y 130.186,Z 509.512,A -85,B 0,C 180,E1 -25866.427,E2 -25866.427} C_VEL
LIN {X 0,Y 137.417,Z 501.862,A -85,B 0,C 180,E1 -25871.671,E2 -25871.671} C_VEL
LIN {X 0,Y 144.515,Z 493.699,A -85,B 0,C 180,E1 -25875.832,E2 -25875.832} C_VEL
LIN {X 0,Y 151.827,Z 484.386,A -85,B 0,C 180,E1 -25879.437,E2 -25879.437} C_VEL
LIN {X 0,Y 159.307,Z 473.753,A -85,B 0,C 180,E1 -25882.567,E2 -25882.567} C_VEL
LIN {X 0,Y 161.562,Z 470.182,A -85,B 0,C 180,E1 -25883.458,E2 -25883.458} C_VEL
LIN {X 0,Y 162.24,Z 464.318,A -85,B 0,C 180,E1 -25886.382,E2 -25886.382} C_VEL
LIN {X 0,Y 161.995,Z 460.584,A -85,B 0,C 180,E1 -25888.627,E2 -25888.627} C_VEL
LIN {X 0,Y 161.015,Z 454.785,A -85,B 0,C 180,E1 -25892.598,E2 -25892.598} C_VEL
LIN {X 0,Y 160.246,Z 451.136,A -85,B 0,C 180,E1 -25895.377,E2 -25895.377} C_VEL
LIN {X 0,Y 158.659,Z 445.519,A -85,B 0,C 180,E1 -25900.596,E2 -25900.596} C_VEL
LIN {X 0,Y 157.618,Z 442.224,A -85,B 0,C 180,E1 -25904.482,E2 -25904.482} C_VEL
LIN {X 0,Y 156.668,Z 438.849,A -85,B 0,C 180,E1 -25909.663,E2 -25909.663} C_VEL
LIN {X 0,Y 156.285,Z 437.819,A -85,B 0,C 180,E1 -25912.246,E2 -25912.246} C_VEL
LIN {X 0,Y 156.23,Z 436.074,A -85,B 0,C 180,E1 -25920,E2 -25920} C_VEL
LIN {X 0,Y 156.455,Z 437.573,A -85,B 0,C 180,E1 -25925.154,E2 -25925.154} C_VEL
LIN {X 0,Y 156.874,Z 438.658,A -85,B 0,C 180,E1 -25927.724,E2 -25927.724} C_VEL
LIN {X 0,Y 157.356,Z 441.698,A -85,B 0,C 180,E1 -25931.593,E2 -25931.593} C_VEL
LIN {X 0,Y 158.098,Z 445.401,A -85,B 0,C 180,E1 -25935.469,E2 -25935.469} C_VEL
LIN {X 0,Y 158.701,Z 448.416,A -85,B 0,C 180,E1 -25938.058,E2 -25938.058} C_VEL
LIN {X 0,Y 159.483,Z 454.338,A -85,B 0,C 180,E1 -25942.272,E2 -25942.272} C_VEL
LIN {X 0,Y 160.14,Z 461.043,A -85,B 0,C 180,E1 -25946.37,E2 -25946.37} C_VEL
LIN {X 0,Y 160.352,Z 466.912,A -85,B 0,C 180,E1 -25949.542,E2 -25949.542} C_VEL
LIN {X 0,Y 159.919,Z 470.442,A -85,B 0,C 180,E1 -25951.089,E2 -25951.089} C_VEL
LIN {X 0,Y 157.92,Z 477.937,A -85,B 0,C 180,E1 -25954.02,E2 -25954.02} C_VEL
LIN {X 0,Y 155.358,Z 485.222,A -85,B 0,C 180,E1 -25956.861,E2 -25956.861} C_VEL
LIN {X 0,Y 153.407,Z 488.349,A -85,B 0,C 180,E1 -25957.791,E2 -25957.791} C_VEL
LIN {X 0,Y 145.174,Z 499.223,A -85,B 0,C 180,E1 -25961.38,E2 -25961.38} C_VEL
LIN {X 0,Y 138.717,Z 507.08,A -85,B 0,C 180,E1 -25964.824,E2 -25964.824} C_VEL
LIN {X 0,Y 131.069,Z 515.855,A -85,B 0,C 180,E1 -25969.953,E2 -25969.953} C_VEL
LIN {X 0,Y 124.394,Z 522.905,A -85,B 0,C 180,E1 -25975.601,E2 -25975.601} C_VEL
LIN {X 0,Y 119.177,Z 528.475,A -85,B 0,C 180,E1 -25981.853,E2 -25981.853} C_VEL
LIN {X 0,Y 115.373,Z 532.705,A -85,B 0,C 180,E1 -25988.564,E2 -25988.564} C_VEL
LIN {X 0,Y 113.046,Z 535.69,A -85,B 0,C 180,E1 -25995.602,E2 -25995.602} C_VEL
LIN {X 0,Y 112.27,Z 537.497,A -85,B 0,C 180,E1 -26002.809,E2 -26002.809} C_VEL
LIN {X 0,Y 112.458,Z 538.106,A -85,B 0,C 180,E1 -26009.197,E2 -26009.197} C_VEL
LIN {X 0,Y 112.34,Z 537.96,A -85,B 0,C 180,E1 -26013.588,E2 -26013.588} C_VEL
LIN {X 0,Y 112.518,Z 536.709,A -85,B 0,C 180,E1 -26020.802,E2 -26020.802} C_VEL
LIN {X 0,Y 113.992,Z 534.292,A -85,B 0,C 180,E1 -26027.956,E2 -26027.956} C_VEL
LIN {X 0,Y 117.089,Z 530.677,A -85,B 0,C 180,E1 -26034.846,E2 -26034.846} C_VEL
LIN {X 0,Y 121.604,Z 525.769,A -85,B 0,C 180,E1 -26041.344,E2 -26041.344} C_VEL
LIN {X 0,Y 127.553,Z 519.446,A -85,B 0,C 180,E1 -26047.309,E2 -26047.309} C_VEL
LIN {X 0,Y 134.771,Z 511.535,A -85,B 0,C 180,E1 -26052.683,E2 -26052.683} C_VEL
LIN {X 0,Y 141.858,Z 503.131,A -85,B 0,C 180,E1 -26056.951,E2 -26056.951} C_VEL
LIN {X 0,Y 149.811,Z 493.036,A -85,B 0,C 180,E1 -26060.721,E2 -26060.721} C_VEL
LIN {X 0,Y 154.652,Z 486.325,A -85,B 0,C 180,E1 -26062.682,E2 -26062.682} C_VEL
LIN {X 0,Y 156.401,Z 482.188,A -85,B 0,C 180,E1 -26064.256,E2 -26064.256} C_VEL
LIN {X 0,Y 158.795,Z 474.457,A -85,B 0,C 180,E1 -26067.238,E2 -26067.238} C_VEL
LIN {X 0,Y 160.143,Z 468.333,A -85,B 0,C 180,E1 -26069.69,E2 -26069.69} C_VEL
LIN {X 0,Y 160.103,Z 462.139,A -85,B 0,C 180,E1 -26072.905,E2 -26072.905} C_VEL
LIN {X 0,Y 159.586,Z 455.77,A -85,B 0,C 180,E1 -26076.65,E2 -26076.65} C_VEL
LIN {X 0,Y 159.082,Z 451.689,A -85,B 0,C 180,E1 -26079.303,E2 -26079.303} C_VEL
LIN {X 0,Y 158.287,Z 446.971,A -85,B 0,C 180,E1 -26082.945,E2 -26082.945} C_VEL
LIN {X 0,Y 157.437,Z 442.554,A -85,B 0,C 180,E1 -26087.103,E2 -26087.103} C_VEL
LIN {X 0,Y 157.014,Z 440.018,A -85,B 0,C 180,E1 -26089.979,E2 -26089.979} C_VEL
LIN {X 0,Y 156.666,Z 438.456,A -85,B 0,C 180,E1 -26092.266,E2 -26092.266} C_VEL
LIN {X 0,Y 156.045,Z 436.628,A -85,B 0,C 180,E1 -26096.997,E2 -26096.997} C_VEL
LIN {X 0,Y 155.673,Z 436.891,A -85,B 0,C 180,E1 -26098.426,E2 -26098.426} C_VEL
LIN {X 0,Y 154.602,Z 438.678,A -85,B 0,C 180,E1 -26100.238,E2 -26100.238} C_VEL
LIN {X 0,Y 152.771,Z 442.051,A -85,B 0,C 180,E1 -26102.947,E2 -26102.947} C_VEL
LIN {X 0,Y 152.397,Z 442.967,A -85,B 0,C 180,E1 -26104.428,E2 -26104.428} C_VEL
LIN {X 0,Y 152.657,Z 443.851,A -85,B 0,C 180,E1 -26107.939,E2 -26107.939} C_VEL
LIN {X 0,Y 152.984,Z 444.952,A -85,B 0,C 180,E1 -26110.589,E2 -26110.589} C_VEL
LIN {X 0,Y 153.837,Z 448.731,A -85,B 0,C 180,E1 -26116.384,E2 -26116.384} C_VEL
LIN {X 0,Y 154.6,Z 451.786,A -85,B 0,C 180,E1 -26119.935,E2 -26119.935} C_VEL
LIN {X 0,Y 155.524,Z 456.049,A -85,B 0,C 180,E1 -26123.998,E2 -26123.998} C_VEL
LIN {X 0,Y 156.352,Z 461.223,A -85,B 0,C 180,E1 -26128.163,E2 -26128.163} C_VEL
LIN {X 0,Y 156.801,Z 466.137,A -85,B 0,C 180,E1 -26131.612,E2 -26131.612} C_VEL
LIN {X 0,Y 156.55,Z 469.808,A -85,B 0,C 180,E1 -26133.758,E2 -26133.758} C_VEL
LIN {X 0,Y 156.07,Z 472.347,A -85,B 0,C 180,E1 -26135.062,E2 -26135.062} C_VEL
LIN {X 0,Y 148.385,Z 482.957,A -85,B 0,C 180,E1 -26138.005,E2 -26138.005} C_VEL
LIN {X 0,Y 142.037,Z 491.054,A -85,B 0,C 180,E1 -26141.01,E2 -26141.01} C_VEL
LIN {X 0,Y 134.348,Z 499.738,A -85,B 0,C 180,E1 -26145.071,E2 -26145.071} C_VEL
LIN {X 0,Y 128.307,Z 506.005,A -85,B 0,C 180,E1 -26148.904,E2 -26148.904} C_VEL
LIN {X 0,Y 121.178,Z 512.888,A -85,B 0,C 180,E1 -26154.55,E2 -26154.55} C_VEL
LIN {X 0,Y 115.361,Z 518.276,A -85,B 0,C 180,E1 -26160.83,E2 -26160.83} C_VEL
LIN {X 0,Y 110.78,Z 522.335,A -85,B 0,C 180,E1 -26167.625,E2 -26167.625} C_VEL
LIN {X 0,Y 107.678,Z 525.172,A -85,B 0,C 180,E1 -26174.865,E2 -26174.865} C_VEL
LIN {X 0,Y 106.03,Z 526.862,A -85,B 0,C 180,E1 -26182.381,E2 -26182.381} C_VEL
LIN {X 0,Y 105.578,Z 527.446,A -85,B 0,C 180,E1 -26189.998,E2 -26189.998} C_VEL
LIN {X 0,Y 106.029,Z 526.892,A -85,B 0,C 180,E1 -26197.616,E2 -26197.616} C_VEL
LIN {X 0,Y 107.66,Z 525.243,A -85,B 0,C 180,E1 -26205.135,E2 -26205.135} C_VEL
LIN {X 0,Y 110.723,Z 522.444,A -85,B 0,C 180,E1 -26212.384,E2 -26212.384} C_VEL
LIN {X 0,Y 115.305,Z 518.419,A -85,B 0,C 180,E1 -26219.182,E2 -26219.182} C_VEL
LIN {X 0,Y 121.073,Z 513.078,A -85,B 0,C 180,E1 -26225.482,E2 -26225.482} C_VEL
LIN {X 0,Y 128.237,Z 506.247,A -85,B 0,C 180,E1 -26231.12,E2 -26231.12} C_VEL
LIN {X 0,Y 136.392,Z 497.71,A -85,B 0,C 180,E1 -26236.168,E2 -26236.168} C_VEL
LIN {X 0,Y 144.278,Z 488.619,A -85,B 0,C 180,E1 -26240.102,E2 -26240.102} C_VEL
LIN {X 0,Y 151.328,Z 479.369,A -85,B 0,C 180,E1 -26243.236,E2 -26243.236} C_VEL
LIN {X 0,Y 156.031,Z 472.75,A -85,B 0,C 180,E1 -26244.979,E2 -26244.979} C_VEL
LIN {X 0,Y 156.627,Z 470.209,A -85,B 0,C 180,E1 -26246.214,E2 -26246.214} C_VEL
LIN {X 0,Y 156.964,Z 466.592,A -85,B 0,C 180,E1 -26248.288,E2 -26248.288} C_VEL
LIN {X 0,Y 156.46,Z 461.557,A -85,B 0,C 180,E1 -26251.858,E2 -26251.858} C_VEL
LIN {X 0,Y 155.707,Z 456.285,A -85,B 0,C 180,E1 -26256.032,E2 -26256.032} C_VEL
LIN {X 0,Y 154.487,Z 450.854,A -85,B 0,C 180,E1 -26261.431,E2 -26261.431} C_VEL
LIN {X 0,Y 153.943,Z 448.612,A -85,B 0,C 180,E1 -26264.102,E2 -26264.102} C_VEL
LIN {X 0,Y 153.149,Z 445.25,A -85,B 0,C 180,E1 -26269.423,E2 -26269.423} C_VEL
LIN {X 0,Y 152.848,Z 444.117,A -85,B 0,C 180,E1 -26272.071,E2 -26272.071} C_VEL
LIN {X 0,Y 152.917,Z 442.381,A -85,B 0,C 180,E1 -26280,E2 -26280} C_VEL
LIN {X 0,Y 153.094,Z 443.906,A -85,B 0,C 180,E1 -26285.268,E2 -26285.268} C_VEL
LIN {X 0,Y 153.397,Z 445.156,A -85,B 0,C 180,E1 -26287.9,E2 -26287.9} C_VEL
LIN {X 0,Y 153.948,Z 449.386,A -85,B 0,C 180,E1 -26293.194,E2 -26293.194} C_VEL
LIN {X 0,Y 154.492,Z 453.624,A -85,B 0,C 180,E1 -26297.197,E2 -26297.197} C_VEL
LIN {X 0,Y 154.917,Z 459.033,A -85,B 0,C 180,E1 -26301.28,E2 -26301.28} C_VEL
LIN {X 0,Y 155.195,Z 464.864,A -85,B 0,C 180,E1 -26305.085,E2 -26305.085} C_VEL
LIN {X 0,Y 155.213,Z 469.604,A -85,B 0,C 180,E1 -26307.851,E2 -26307.851} C_VEL
LIN {X 0,Y 154.822,Z 472.654,A -85,B 0,C 180,E1 -26309.41,E2 -26309.41} C_VEL
LIN {X 0,Y 153.08,Z 478.651,A -85,B 0,C 180,E1 -26311.925,E2 -26311.925} C_VEL
LIN {X 0,Y 149.96,Z 486.676,A -85,B 0,C 180,E1 -26315.197,E2 -26315.197} C_VEL
LIN {X 0,Y 142.953,Z 495.937,A -85,B 0,C 180,E1 -26318.132,E2 -26318.132} C_VEL
LIN {X 0,Y 134.821,Z 505.482,A -85,B 0,C 180,E1 -26322.029,E2 -26322.029} C_VEL
LIN {X 0,Y 127.565,Z 513.458,A -85,B 0,C 180,E1 -26326.477,E2 -26326.477} C_VEL
LIN {X 0,Y 120.177,Z 520.914,A -85,B 0,C 180,E1 -26332.119,E2 -26332.119} C_VEL
LIN {X 0,Y 114.172,Z 526.853,A -85,B 0,C 180,E1 -26338.453,E2 -26338.453} C_VEL
LIN {X 0,Y 110.61,Z 530.399,A -85,B 0,C 180,E1 -26343.593,E2 -26343.593} C_VEL
LIN {X 0,Y 107.2,Z 533.996,A -85,B 0,C 180,E1 -26350.866,E2 -26350.866} C_VEL
LIN {X 0,Y 105.493,Z 536.39,A -85,B 0,C 180,E1 -26358.473,E2 -26358.473} C_VEL
LIN {X 0,Y 105.238,Z 537.618,A -85,B 0,C 180,E1 -26366.172,E2 -26366.172} C_VEL
LIN {X 0,Y 105.419,Z 537.788,A -85,B 0,C 180,E1 -26370.002,E2 -26370.002} C_VEL
LIN {X 0,Y 105.239,Z 537.612,A -85,B 0,C 180,E1 -26373.831,E2 -26373.831} C_VEL
LIN {X 0,Y 105.505,Z 536.358,A -85,B 0,C 180,E1 -26381.529,E2 -26381.529} C_VEL
LIN {X 0,Y 107.204,Z 533.941,A -85,B 0,C 180,E1 -26389.136,E2 -26389.136} C_VEL
LIN {X 0,Y 110.597,Z 530.324,A -85,B 0,C 180,E1 -26396.414,E2 -26396.414} C_VEL
LIN {X 0,Y 115.518,Z 525.415,A -85,B 0,C 180,E1 -26403.201,E2 -26403.201} C_VEL
LIN {X 0,Y 121.934,Z 519.094,A -85,B 0,C 180,E1 -26409.349,E2 -26409.349} C_VEL
LIN {X 0,Y 129.553,Z 511.179,A -85,B 0,C 180,E1 -26414.849,E2 -26414.849} C_VEL
LIN {X 0,Y 137.065,Z 502.778,A -85,B 0,C 180,E1 -26419.142,E2 -26419.142} C_VEL
LIN {X 0,Y 145.379,Z 492.682,A -85,B 0,C 180,E1 -26422.908,E2 -26422.908} C_VEL
LIN {X 0,Y 149.914,Z 486.491,A -85,B 0,C 180,E1 -26424.782,E2 -26424.782} C_VEL
LIN {X 0,Y 152.967,Z 478.449,A -85,B 0,C 180,E1 -26428.088,E2 -26428.088} C_VEL
LIN {X 0,Y 154.734,Z 472.36,A -85,B 0,C 180,E1 -26430.633,E2 -26430.633} C_VEL
LIN {X 0,Y 155.082,Z 467.824,A -85,B 0,C 180,E1 -26433.052,E2 -26433.052} C_VEL
LIN {X 0,Y 154.994,Z 462.005,A -85,B 0,C 180,E1 -26436.594,E2 -26436.594} C_VEL
LIN {X 0,Y 154.695,Z 456.864,A -85,B 0,C 180,E1 -26440.079,E2 -26440.079} C_VEL
LIN {X 0,Y 154.112,Z 451.939,A -85,B 0,C 180,E1 -26444.121,E2 -26444.121} C_VEL
LIN {X 0,Y 153.624,Z 447.997,A -85,B 0,C 180,E1 -26448.12,E2 -26448.12} C_VEL
LIN {X 0,Y 153.217,Z 444.928,A -85,B 0,C 180,E1 -26452.091,E2 -26452.091} C_VEL
LIN {X 0,Y 152.923,Z 443.65,A -85,B 0,C 180,E1 -26454.726,E2 -26454.726} C_VEL
LIN {X 0,Y 152.818,Z 441.974,A -85,B 0,C 180,E1 -26460,E2 -26460} C_VEL
LIN {X 0,Y 152.397,Z 442.967,A -85,B 0,C 180,E1 -26464.428,E2 -26464.428} C_VEL
LIN {X 0,Y 152.139,Z 444.165,A -85,B 0,C 180,E1 -26466.602,E2 -26466.602} C_VEL
LIN {X 0,Y 151.458,Z 446.29,A -85,B 0,C 180,E1 -26468.684,E2 -26468.684} C_VEL
LIN {X 0,Y 149.621,Z 453.023,A -85,B 0,C 180,E1 -26474.203,E2 -26474.203} C_VEL
LIN {X 0,Y 149.642,Z 454.241,A -85,B 0,C 180,E1 -26475.669,E2 -26475.669} C_VEL
LIN {X 0,Y 150.219,Z 456.957,A -85,B 0,C 180,E1 -26479.117,E2 -26479.117} C_VEL
LIN {X 0,Y 150.831,Z 461.045,A -85,B 0,C 180,E1 -26483.332,E2 -26483.332} C_VEL
LIN {X 0,Y 151.394,Z 466.674,A -85,B 0,C 180,E1 -26488.111,E2 -26488.111} C_VEL
LIN {X 0,Y 151.507,Z 470.128,A -85,B 0,C 180,E1 -26490.682,E2 -26490.682} C_VEL
LIN {X 0,Y 150.991,Z 474.056,A -85,B 0,C 180,E1 -26493.087,E2 -26493.087} C_VEL
LIN {X 0,Y 148.587,Z 477.573,A -85,B 0,C 180,E1 -26494.132,E2 -26494.132} C_VEL
LIN {X 0,Y 142.686,Z 485.189,A -85,B 0,C 180,E1 -26496.424,E2 -26496.424} C_VEL
LIN {X 0,Y 135.098,Z 494.084,A -85,B 0,C 180,E1 -26499.884,E2 -26499.884} C_VEL
LIN {X 0,Y 127.227,Z 502.293,A -85,B 0,C 180,E1 -26504.099,E2 -26504.099} C_VEL
LIN {X 0,Y 119.11,Z 509.994,A -85,B 0,C 180,E1 -26509.528,E2 -26509.528} C_VEL
LIN {X 0,Y 112.188,Z 516.106,A -85,B 0,C 180,E1 -26515.679,E2 -26515.679} C_VEL
LIN {X 0,Y 106.463,Z 520.818,A -85,B 0,C 180,E1 -26522.476,E2 -26522.476} C_VEL
LIN {X 0,Y 102.376,Z 524.248,A -85,B 0,C 180,E1 -26529.924,E2 -26529.924} C_VEL
LIN {X 0,Y 99.72,Z 526.505,A -85,B 0,C 180,E1 -26537.792,E2 -26537.792} C_VEL
LIN {X 0,Y 98.586,Z 527.66,A -85,B 0,C 180,E1 -26546.416,E2 -26546.416} C_VEL
LIN {X 0,Y 98.612,Z 527.652,A -85,B 0,C 180,E1 -26554.085,E2 -26554.085} C_VEL
LIN {X 0,Y 99.716,Z 526.555,A -85,B 0,C 180,E1 -26562.205,E2 -26562.205} C_VEL
LIN {X 0,Y 102.301,Z 524.339,A -85,B 0,C 180,E1 -26570.088,E2 -26570.088} C_VEL
LIN {X 0,Y 106.411,Z 520.941,A -85,B 0,C 180,E1 -26577.535,E2 -26577.535} C_VEL
LIN {X 0,Y 112.099,Z 516.269,A -85,B 0,C 180,E1 -26584.348,E2 -26584.348} C_VEL
LIN {X 0,Y 119.034,Z 510.206,A -85,B 0,C 180,E1 -26590.499,E2 -26590.499} C_VEL
LIN {X 0,Y 127.15,Z 502.555,A -85,B 0,C 180,E1 -26595.933,E2 -26595.933} C_VEL
LIN {X 0,Y 134.992,Z 494.392,A -85,B 0,C 180,E1 -26600.165,E2 -26600.165} C_VEL
LIN {X 0,Y 142.375,Z 485.816,A -85,B 0,C 180,E1 -26603.506,E2 -26603.506} C_VEL
LIN {X 0,Y 149.781,Z 476.212,A -85,B 0,C 180,E1 -26606.392,E2 -26606.392} C_VEL
LIN {X 0,Y 151.035,Z 474.449,A -85,B 0,C 180,E1 -26606.883,E2 -26606.883} C_VEL
LIN {X 0,Y 151.615,Z 470.408,A -85,B 0,C 180,E1 -26609.343,E2 -26609.343} C_VEL
LIN {X 0,Y 151.335,Z 465.067,A -85,B 0,C 180,E1 -26613.449,E2 -26613.449} C_VEL
LIN {X 0,Y 151.003,Z 461.278,A -85,B 0,C 180,E1 -26616.696,E2 -26616.696} C_VEL
LIN {X 0,Y 150.369,Z 457.23,A -85,B 0,C 180,E1 -26620.903,E2 -26620.903} C_VEL
LIN {X 0,Y 149.955,Z 454.929,A -85,B 0,C 180,E1 -26623.668,E2 -26623.668} C_VEL
LIN {X 0,Y 149.342,Z 451.527,A -85,B 0,C 180,E1 -26629.15,E2 -26629.15} C_VEL
LIN {X 0,Y 149.14,Z 450.302,A -85,B 0,C 180,E1 -26631.873,E2 -26631.873} C_VEL
LIN {X 0,Y 149.348,Z 448.554,A -85,B 0,C 180,E1 -26640,E2 -26640} C_VEL
LIN {X 0,Y 149.457,Z 450.131,A -85,B 0,C 180,E1 -26645.396,E2 -26645.396} C_VEL
LIN {X 0,Y 149.631,Z 451.536,A -85,B 0,C 180,E1 -26648.1,E2 -26648.1} C_VEL
LIN {X 0,Y 149.891,Z 454.657,A -85,B 0,C 180,E1 -26652.18,E2 -26652.18} C_VEL
LIN {X 0,Y 150.139,Z 458.731,A -85,B 0,C 180,E1 -26656.311,E2 -26656.311} C_VEL
LIN {X 0,Y 150.27,Z 463.16,A -85,B 0,C 180,E1 -26659.897,E2 -26659.897} C_VEL
LIN {X 0,Y 150.232,Z 469.272,A -85,B 0,C 180,E1 -26664.163,E2 -26664.163} C_VEL
LIN {X 0,Y 149.922,Z 473.905,A -85,B 0,C 180,E1 -26667.044,E2 -26667.044} C_VEL
LIN {X 0,Y 149.211,Z 476.987,A -85,B 0,C 180,E1 -26668.6,E2 -26668.6} C_VEL
LIN {X 0,Y 146.313,Z 484.531,A -85,B 0,C 180,E1 -26671.895,E2 -26671.895} C_VEL
LIN {X 0,Y 144.601,Z 488.182,A -85,B 0,C 180,E1 -26673.444,E2 -26673.444} C_VEL
LIN {X 0,Y 136.145,Z 498.526,A -85,B 0,C 180,E1 -26676.859,E2 -26676.859} C_VEL
LIN {X 0,Y 127.895,Z 507.551,A -85,B 0,C 180,E1 -26680.874,E2 -26680.874} C_VEL
LIN {X 0,Y 120.371,Z 515.15,A -85,B 0,C 180,E1 -26685.524,E2 -26685.524} C_VEL
LIN {X 0,Y 112.839,Z 522.204,A -85,B 0,C 180,E1 -26691.478,E2 -26691.478} C_VEL
LIN {X 0,Y 106.719,Z 527.772,A -85,B 0,C 180,E1 -26698.21,E2 -26698.21} C_VEL
LIN {X 0,Y 102.122,Z 532.001,A -85,B 0,C 180,E1 -26705.614,E2 -26705.614} C_VEL
LIN {X 0,Y 99.224,Z 534.988,A -85,B 0,C 180,E1 -26713.544,E2 -26713.544} C_VEL
LIN {X 0,Y 98.12,Z 536.798,A -85,B 0,C 180,E1 -26721.766,E2 -26721.766} C_VEL
LIN {X 0,Y 98.123,Z 537.268,A -85,B 0,C 180,E1 -26725.894,E2 -26725.894} C_VEL
LIN {X 0,Y 98.331,Z 537.441,A -85,B 0,C 180,E1 -26730.002,E2 -26730.002} C_VEL
LIN {X 0,Y 98.124,Z 537.262,A -85,B 0,C 180,E1 -26734.109,E2 -26734.109} C_VEL
LIN {X 0,Y 98.492,Z 536.007,A -85,B 0,C 180,E1 -26742.363,E2 -26742.363} C_VEL
LIN {X 0,Y 100.47,Z 533.589,A -85,B 0,C 180,E1 -26750.474,E2 -26750.474} C_VEL
LIN {X 0,Y 104.185,Z 529.969,A -85,B 0,C 180,E1 -26758.179,E2 -26758.179} C_VEL
LIN {X 0,Y 109.557,Z 525.061,A -85,B 0,C 180,E1 -26765.266,E2 -26765.266} C_VEL
LIN {X 0,Y 116.482,Z 518.741,A -85,B 0,C 180,E1 -26771.584,E2 -26771.584} C_VEL
LIN {X 0,Y 124.547,Z 510.824,A -85,B 0,C 180,E1 -26777.189,E2 -26777.189} C_VEL
LIN {X 0,Y 132.496,Z 502.425,A -85,B 0,C 180,E1 -26781.481,E2 -26781.481} C_VEL
LIN {X 0,Y 141.167,Z 492.328,A -85,B 0,C 180,E1 -26785.232,E2 -26785.232} C_VEL
LIN {X 0,Y 144.583,Z 487.961,A -85,B 0,C 180,E1 -26786.551,E2 -26786.551} C_VEL
LIN {X 0,Y 147.826,Z 480.402,A -85,B 0,C 180,E1 -26789.826,E2 -26789.826} C_VEL
LIN {X 0,Y 149.5,Z 475.587,A -85,B 0,C 180,E1 -26791.96,E2 -26791.96} C_VEL
LIN {X 0,Y 150.053,Z 470.251,A -85,B 0,C 180,E1 -26795.069,E2 -26795.069} C_VEL
LIN {X 0,Y 150.119,Z 463.856,A -85,B 0,C 180,E1 -26799.446,E2 -26799.446} C_VEL
LIN {X 0,Y 150.014,Z 459.925,A -85,B 0,C 180,E1 -26802.534,E2 -26802.534} C_VEL
LIN {X 0,Y 149.817,Z 455.699,A -85,B 0,C 180,E1 -26806.435,E2 -26806.435} C_VEL
LIN {X 0,Y 149.512,Z 452.072,A -85,B 0,C 180,E1 -26810.805,E2 -26810.805} C_VEL
LIN {X 0,Y 149.3,Z 449.885,A -85,B 0,C 180,E1 -26814.598,E2 -26814.598} C_VEL
LIN {X 0,Y 149.265,Z 448.167,A -85,B 0,C 180,E1 -26820,E2 -26820} C_VEL
LIN {X 0,Y 148.975,Z 450.027,A -85,B 0,C 180,E1 -26828.137,E2 -26828.137} C_VEL
LIN {X 0,Y 149.186,Z 451.239,A -85,B 0,C 180,E1 -26830.862,E2 -26830.862} C_VEL
LIN {X 0,Y 149.642,Z 454.241,A -85,B 0,C 180,E1 -26835.669,E2 -26835.669} C_VEL
LIN {X 0,Y 149.641,Z 456.332,A -85,B 0,C 180,E1 -26837.781,E2 -26837.781} C_VEL
LIN {X 0,Y 148.959,Z 459.266,A -85,B 0,C 180,E1 -26839.748,E2 -26839.748} C_VEL
LIN {X 0,Y 146.389,Z 468.09,A -85,B 0,C 180,E1 -26844.904,E2 -26844.904} C_VEL
LIN {X 0,Y 146.198,Z 469.912,A -85,B 0,C 180,E1 -26846.314,E2 -26846.314} C_VEL
LIN {X 0,Y 146.103,Z 474.518,A -85,B 0,C 180,E1 -26850.018,E2 -26850.018} C_VEL
LIN {X 0,Y 145.795,Z 476.183,A -85,B 0,C 180,E1 -26851.168,E2 -26851.168} C_VEL
LIN {X 0,Y 144.728,Z 477.923,A -85,B 0,C 180,E1 -26851.808,E2 -26851.808} C_VEL
LIN {X 0,Y 138.252,Z 485.908,A -85,B 0,C 180,E1 -26854.18,E2 -26854.18} C_VEL
LIN {X 0,Y 130.66,Z 494.434,A -85,B 0,C 180,E1 -26857.496,E2 -26857.496} C_VEL
LIN {X 0,Y 122.383,Z 502.643,A -85,B 0,C 180,E1 -26861.706,E2 -26861.706} C_VEL
LIN {X 0,Y 113.786,Z 510.344,A -85,B 0,C 180,E1 -26867.2,E2 -26867.2} C_VEL
LIN {X 0,Y 106.371,Z 516.457,A -85,B 0,C 180,E1 -26873.511,E2 -26873.511} C_VEL
LIN {X 0,Y 100.2,Z 521.168,A -85,B 0,C 180,E1 -26880.593,E2 -26880.593} C_VEL
LIN {X 0,Y 95.714,Z 524.598,A -85,B 0,C 180,E1 -26888.459,E2 -26888.459} C_VEL
LIN {X 0,Y 92.779,Z 526.854,A -85,B 0,C 180,E1 -26896.863,E2 -26896.863} C_VEL
LIN {X 0,Y 91.55,Z 527.989,A -85,B 0,C 180,E1 -26905.595,E2 -26905.595} C_VEL
LIN {X 0,Y 91.55,Z 527.999,A -85,B 0,C 180,E1 -26914.401,E2 -26914.401} C_VEL
LIN {X 0,Y 92.773,Z 526.904,A -85,B 0,C 180,E1 -26923.134,E2 -26923.134} C_VEL
LIN {X 0,Y 95.649,Z 524.687,A -85,B 0,C 180,E1 -26931.552,E2 -26931.552} C_VEL
LIN {X 0,Y 100.151,Z 521.289,A -85,B 0,C 180,E1 -26939.419,E2 -26939.419} C_VEL
LIN {X 0,Y 106.27,Z 516.618,A -85,B 0,C 180,E1 -26946.525,E2 -26946.525} C_VEL
LIN {X 0,Y 113.705,Z 510.554,A -85,B 0,C 180,E1 -26952.834,E2 -26952.834} C_VEL
LIN {X 0,Y 122.3,Z 502.903,A -85,B 0,C 180,E1 -26958.333,E2 -26958.333} C_VEL
LIN {X 0,Y 130.561,Z 494.738,A -85,B 0,C 180,E1 -26962.557,E2 -26962.557} C_VEL
LIN {X 0,Y 139.234,Z 485.034,A -85,B 0,C 180,E1 -26966.272,E2 -26966.272} C_VEL
LIN {X 0,Y 145.864,Z 476.567,A -85,B 0,C 180,E1 -26968.782,E2 -26968.782} C_VEL
LIN {X 0,Y 146.298,Z 473.096,A -85,B 0,C 180,E1 -26971.289,E2 -26971.289} C_VEL
LIN {X 0,Y 146.209,Z 467.706,A -85,B 0,C 180,E1 -26975.962,E2 -26975.962} C_VEL
LIN {X 0,Y 145.992,Z 464.57,A -85,B 0,C 180,E1 -26979.121,E2 -26979.121} C_VEL
LIN {X 0,Y 145.66,Z 461.143,A -85,B 0,C 180,E1 -26983.172,E2 -26983.172} C_VEL
LIN {X 0,Y 145.423,Z 459.226,A -85,B 0,C 180,E1 -26986.016,E2 -26986.016} C_VEL
LIN {X 0,Y 145.274,Z 457.63,A -85,B 0,C 180,E1 -26988.842,E2 -26988.842} C_VEL
LIN {X 0,Y 145.162,Z 456.362,A -85,B 0,C 180,E1 -26991.648,E2 -26991.648} C_VEL
LIN {X 0,Y 145.153,Z 455.046,A -85,B 0,C 180,E1 -26997.224,E2 -26997.224} C_VEL
LIN {X 0,Y 145.53,Z 454.582,A -85,B 0,C 180,E1 -27000,E2 -27000} C_VEL
LIN {X 0,Y 145.552,Z 456.23,A -85,B 0,C 180,E1 -27005.541,E2 -27005.541} C_VEL
LIN {X 0,Y 145.616,Z 458.844,A -85,B 0,C 180,E1 -27009.889,E2 -27009.889} C_VEL
LIN {X 0,Y 145.67,Z 462.293,A -85,B 0,C 180,E1 -27013.959,E2 -27013.959} C_VEL
LIN {X 0,Y 145.58,Z 466.999,A -85,B 0,C 180,E1 -27018.288,E2 -27018.288} C_VEL
LIN {X 0,Y 145.156,Z 473.359,A -85,B 0,C 180,E1 -27023.089,E2 -27023.089} C_VEL
LIN {X 0,Y 144.391,Z 478.584,A -85,B 0,C 180,E1 -27026.466,E2 -27026.466} C_VEL
LIN {X 0,Y 141.988,Z 484.468,A -85,B 0,C 180,E1 -27029.236,E2 -27029.236} C_VEL
LIN {X 0,Y 139.8,Z 488.934,A -85,B 0,C 180,E1 -27031.284,E2 -27031.284} C_VEL
LIN {X 0,Y 131.967,Z 498.177,A -85,B 0,C 180,E1 -27034.367,E2 -27034.367} C_VEL
LIN {X 0,Y 123.266,Z 507.252,A -85,B 0,C 180,E1 -27038.38,E2 -27038.38} C_VEL
LIN {X 0,Y 115.354,Z 514.8,A -85,B 0,C 180,E1 -27043.023,E2 -27043.023} C_VEL
LIN {X 0,Y 107.3,Z 521.852,A -85,B 0,C 180,E1 -27049.084,E2 -27049.084} C_VEL
LIN {X 0,Y 100.668,Z 527.42,A -85,B 0,C 180,E1 -27056.049,E2 -27056.049} C_VEL
LIN {X 0,Y 95.623,Z 531.65,A -85,B 0,C 180,E1 -27063.835,E2 -27063.835} C_VEL
LIN {X 0,Y 92.366,Z 534.637,A -85,B 0,C 180,E1 -27072.283,E2 -27072.283} C_VEL
LIN {X 0,Y 91.064,Z 536.448,A -85,B 0,C 180,E1 -27081.123,E2 -27081.123} C_VEL
LIN {X 0,Y 91.244,Z 537.093,A -85,B 0,C 180,E1 -27090.002,E2 -27090.002} C_VEL
LIN {X 0,Y 91.083,Z 536.429,A -85,B 0,C 180,E1 -27098.879,E2 -27098.879} C_VEL
LIN {X 0,Y 92.385,Z 534.591,A -85,B 0,C 180,E1 -27107.717,E2 -27107.717} C_VEL
LIN {X 0,Y 95.62,Z 531.581,A -85,B 0,C 180,E1 -27116.169,E2 -27116.169} C_VEL
LIN {X 0,Y 100.648,Z 527.331,A -85,B 0,C 180,E1 -27123.963,E2 -27123.963} C_VEL
LIN {X 0,Y 107.298,Z 521.732,A -85,B 0,C 180,E1 -27130.922,E2 -27130.922} C_VEL
LIN {X 0,Y 115.366,Z 514.642,A -85,B 0,C 180,E1 -27136.975,E2 -27136.975} C_VEL
LIN {X 0,Y 124.456,Z 505.837,A -85,B 0,C 180,E1 -27142.242,E2 -27142.242} C_VEL
LIN {X 0,Y 133.283,Z 496.512,A -85,B 0,C 180,E1 -27146.152,E2 -27146.152} C_VEL
LIN {X 0,Y 139.777,Z 488.681,A -85,B 0,C 180,E1 -27148.735,E2 -27148.735} C_VEL
LIN {X 0,Y 143.586,Z 480.4,A -85,B 0,C 180,E1 -27152.562,E2 -27152.562} C_VEL
LIN {X 0,Y 144.466,Z 477.538,A -85,B 0,C 180,E1 -27154.035,E2 -27154.035} C_VEL
LIN {X 0,Y 145.14,Z 471.686,A -85,B 0,C 180,E1 -27157.96,E2 -27157.96} C_VEL
LIN {X 0,Y 145.444,Z 466.818,A -85,B 0,C 180,E1 -27161.695,E2 -27161.695} C_VEL
LIN {X 0,Y 145.503,Z 462.14,A -85,B 0,C 180,E1 -27166.025,E2 -27166.025} C_VEL
LIN {X 0,Y 145.513,Z 459.564,A -85,B 0,C 180,E1 -27168.861,E2 -27168.861} C_VEL
LIN {X 0,Y 145.464,Z 457.516,A -85,B 0,C 180,E1 -27171.666,E2 -27171.666} C_VEL
LIN {X 0,Y 145.406,Z 455.995,A -85,B 0,C 180,E1 -27174.453,E2 -27174.453} C_VEL
LIN {X 0,Y 145.464,Z 454.212,A -85,B 0,C 180,E1 -27180,E2 -27180} C_VEL
LIN {X 0,Y 145.014,Z 456.094,A -85,B 0,C 180,E1 -27188.36,E2 -27188.36} C_VEL
LIN {X 0,Y 145.132,Z 457.348,A -85,B 0,C 180,E1 -27191.169,E2 -27191.169} C_VEL
LIN {X 0,Y 145.514,Z 460.883,A -85,B 0,C 180,E1 -27196.846,E2 -27196.846} C_VEL
LIN {X 0,Y 145.913,Z 464.944,A -85,B 0,C 180,E1 -27201.591,E2 -27201.591} C_VEL
LIN {X 0,Y 146.203,Z 469.141,A -85,B 0,C 180,E1 -27205.635,E2 -27205.635} C_VEL
LIN {X 0,Y 146.198,Z 469.912,A -85,B 0,C 180,E1 -27206.314,E2 -27206.314} C_VEL
LIN {X 0,Y 145.714,Z 471.929,A -85,B 0,C 180,E1 -27207.602,E2 -27207.602} C_VEL
LIN {X 0,Y 144.059,Z 475.131,A -85,B 0,C 180,E1 -27208.924,E2 -27208.924} C_VEL
LIN {X 0,Y 141.628,Z 478.563,A -85,B 0,C 180,E1 -27209.995,E2 -27209.995} C_VEL
LIN {X 0,Y 135.258,Z 485.783,A -85,B 0,C 180,E1 -27211.798,E2 -27211.798} C_VEL
LIN {X 0,Y 129.936,Z 491.211,A -85,B 0,C 180,E1 -27213.499,E2 -27213.499} C_VEL
LIN {X 0,Y 121.427,Z 499.679,A -85,B 0,C 180,E1 -27217.264,E2 -27217.264} C_VEL
LIN {X 0,Y 113.096,Z 507.056,A -85,B 0,C 180,E1 -27221.778,E2 -27221.778} C_VEL
LIN {X 0,Y 104.511,Z 513.939,A -85,B 0,C 180,E1 -27227.74,E2 -27227.74} C_VEL
LIN {X 0,Y 97.266,Z 519.326,A -85,B 0,C 180,E1 -27234.685,E2 -27234.685} C_VEL
LIN {X 0,Y 91.401,Z 523.384,A -85,B 0,C 180,E1 -27242.523,E2 -27242.523} C_VEL
LIN {X 0,Y 87.269,Z 526.218,A -85,B 0,C 180,E1 -27251.206,E2 -27251.206} C_VEL
LIN {X 0,Y 84.96,Z 527.907,A -85,B 0,C 180,E1 -27260.475,E2 -27260.475} C_VEL
LIN {X 0,Y 84.337,Z 528.487,A -85,B 0,C 180,E1 -27269.998,E2 -27269.998} C_VEL
LIN {X 0,Y 84.958,Z 527.936,A -85,B 0,C 180,E1 -27279.521,E2 -27279.521} C_VEL
LIN {X 0,Y 87.246,Z 526.287,A -85,B 0,C 180,E1 -27288.795,E2 -27288.795} C_VEL
LIN {X 0,Y 91.341,Z 523.488,A -85,B 0,C 180,E1 -27297.492,E2 -27297.492} C_VEL
LIN {X 0,Y 97.192,Z 519.464,A -85,B 0,C 180,E1 -27305.342,E2 -27305.342} C_VEL
LIN {X 0,Y 104.411,Z 514.122,A -85,B 0,C 180,E1 -27312.305,E2 -27312.305} C_VEL
LIN {X 0,Y 113.032,Z 507.288,A -85,B 0,C 180,E1 -27318.253,E2 -27318.253} C_VEL
LIN {X 0,Y 122.554,Z 498.752,A -85,B 0,C 180,E1 -27323.4,E2 -27323.4} C_VEL
LIN {X 0,Y 131.594,Z 489.66,A -85,B 0,C 180,E1 -27327.259,E2 -27327.259} C_VEL
LIN {X 0,Y 139.526,Z 480.527,A -85,B 0,C 180,E1 -27330.217,E2 -27330.217} C_VEL
LIN {X 0,Y 140.67,Z 478.952,A -85,B 0,C 180,E1 -27330.739,E2 -27330.739} C_VEL
LIN {X 0,Y 141.039,Z 475.428,A -85,B 0,C 180,E1 -27333.756,E2 -27333.756} C_VEL
LIN {X 0,Y 141.246,Z 470.916,A -85,B 0,C 180,E1 -27338.088,E2 -27338.088} C_VEL
LIN {X 0,Y 141.104,Z 467.178,A -85,B 0,C 180,E1 -27342.612,E2 -27342.612} C_VEL
LIN {X 0,Y 141.03,Z 465.175,A -85,B 0,C 180,E1 -27345.571,E2 -27345.571} C_VEL
LIN {X 0,Y 140.936,Z 462.263,A -85,B 0,C 180,E1 -27351.396,E2 -27351.396} C_VEL
LIN {X 0,Y 141.058,Z 460.896,A -85,B 0,C 180,E1 -27357.144,E2 -27357.144} C_VEL
LIN {X 0,Y 141.48,Z 460.44,A -85,B 0,C 180,E1 -27360,E2 -27360} C_VEL
LIN {X 0,Y 141.375,Z 462.197,A -85,B 0,C 180,E1 -27365.706,E2 -27365.706} C_VEL
LIN {X 0,Y 141.285,Z 464.775,A -85,B 0,C 180,E1 -27370.026,E2 -27370.026} C_VEL
LIN {X 0,Y 141.041,Z 468.572,A -85,B 0,C 180,E1 -27374.427,E2 -27374.427} C_VEL
LIN {X 0,Y 140.601,Z 472.733,A -85,B 0,C 180,E1 -27378.25,E2 -27378.25} C_VEL
LIN {X 0,Y 139.768,Z 478.759,A -85,B 0,C 180,E1 -27382.984,E2 -27382.984} C_VEL
LIN {X 0,Y 138.962,Z 482.203,A -85,B 0,C 180,E1 -27385.279,E2 -27385.279} C_VEL
LIN {X 0,Y 135.793,Z 488.543,A -85,B 0,C 180,E1 -27388.38,E2 -27388.38} C_VEL
LIN {X 0,Y 134.849,Z 490.23,A -85,B 0,C 180,E1 -27389.197,E2 -27389.197} C_VEL
LIN {X 0,Y 126.723,Z 499.195,A -85,B 0,C 180,E1 -27392.249,E2 -27392.249} C_VEL
LIN {X 0,Y 117.693,Z 508.031,A -85,B 0,C 180,E1 -27396.281,E2 -27396.281} C_VEL
LIN {X 0,Y 110.59,Z 514.45,A -85,B 0,C 180,E1 -27400.309,E2 -27400.309} C_VEL
LIN {X 0,Y 101.978,Z 521.501,A -85,B 0,C 180,E1 -27406.438,E2 -27406.438} C_VEL
LIN {X 0,Y 94.779,Z 527.068,A -85,B 0,C 180,E1 -27413.617,E2 -27413.617} C_VEL
LIN {X 0,Y 89.235,Z 531.298,A -85,B 0,C 180,E1 -27421.802,E2 -27421.802} C_VEL
LIN {X 0,Y 85.558,Z 534.285,A -85,B 0,C 180,E1 -27430.82,E2 -27430.82} C_VEL
LIN {X 0,Y 84.008,Z 536.098,A -85,B 0,C 180,E1 -27440.37,E2 -27440.37} C_VEL
LIN {X 0,Y 84.143,Z 536.745,A -85,B 0,C 180,E1 -27450.002,E2 -27450.002} C_VEL
LIN {X 0,Y 84.024,Z 536.079,A -85,B 0,C 180,E1 -27459.632,E2 -27459.632} C_VEL
LIN {X 0,Y 85.575,Z 534.239,A -85,B 0,C 180,E1 -27469.18,E2 -27469.18} C_VEL
LIN {X 0,Y 89.226,Z 531.228,A -85,B 0,C 180,E1 -27478.205,E2 -27478.205} C_VEL
LIN {X 0,Y 94.758,Z 526.977,A -85,B 0,C 180,E1 -27486.397,E2 -27486.397} C_VEL
LIN {X 0,Y 101.976,Z 521.379,A -85,B 0,C 180,E1 -27493.568,E2 -27493.568} C_VEL
LIN {X 0,Y 110.599,Z 514.289,A -85,B 0,C 180,E1 -27499.691,E2 -27499.691} C_VEL
LIN {X 0,Y 118.941,Z 506.719,A -85,B 0,C 180,E1 -27504.34,E2 -27504.34} C_VEL
LIN {X 0,Y 128.071,Z 497.619,A -85,B 0,C 180,E1 -27508.277,E2 -27508.277} C_VEL
LIN {X 0,Y 134.811,Z 489.97,A -85,B 0,C 180,E1 -27510.837,E2 -27510.837} C_VEL
LIN {X 0,Y 138.657,Z 482.477,A -85,B 0,C 180,E1 -27514.482,E2 -27514.482} C_VEL
LIN {X 0,Y 139.432,Z 479.732,A -85,B 0,C 180,E1 -27516.22,E2 -27516.22} C_VEL
LIN {X 0,Y 140.164,Z 475.33,A -85,B 0,C 180,E1 -27519.453,E2 -27519.453} C_VEL
LIN {X 0,Y 140.697,Z 470.485,A -85,B 0,C 180,E1 -27523.535,E2 -27523.535} C_VEL
LIN {X 0,Y 140.996,Z 467.03,A -85,B 0,C 180,E1 -27527.038,E2 -27527.038} C_VEL
LIN {X 0,Y 141.186,Z 463.571,A -85,B 0,C 180,E1 -27531.412,E2 -27531.412} C_VEL
LIN {X 0,Y 141.246,Z 461.933,A -85,B 0,C 180,E1 -27534.362,E2 -27534.362} C_VEL
LIN {X 0,Y 141.415,Z 460.108,A -85,B 0,C 180,E1 -27540,E2 -27540} C_VEL
LIN {X 0,Y 140.774,Z 461.753,A -85,B 0,C 180,E1 -27547.794,E2 -27547.794} C_VEL
LIN {X 0,Y 140.806,Z 463.313,A -85,B 0,C 180,E1 -27551.517,E2 -27551.517} C_VEL
LIN {X 0,Y 140.859,Z 464.974,A -85,B 0,C 180,E1 -27554.446,E2 -27554.446} C_VEL
LIN {X 0,Y 141.019,Z 467.961,A -85,B 0,C 180,E1 -27558.751,E2 -27558.751} C_VEL
LIN {X 0,Y 141.06,Z 472.2,A -85,B 0,C 180,E1 -27563.49,E2 -27563.49} C_VEL
LIN {X 0,Y 140.879,Z 476.504,A -85,B 0,C 180,E1 -27567.52,E2 -27567.52} C_VEL
LIN {X 0,Y 140.581,Z 478.624,A -85,B 0,C 180,E1 -27569.236,E2 -27569.236} C_VEL
LIN {X 0,Y 139.585,Z 480.187,A -85,B 0,C 180,E1 -27569.843,E2 -27569.843} C_VEL
LIN {X 0,Y 132.959,Z 487.864,A -85,B 0,C 180,E1 -27572.247,E2 -27572.247} C_VEL
LIN {X 0,Y 129.936,Z 491.211,A -85,B 0,C 180,E1 -27573.499,E2 -27573.499} C_VEL
LIN {X 0,Y 126.072,Z 494.846,A -85,B 0,C 180,E1 -27574.719,E2 -27574.719} C_VEL
LIN {X 0,Y 118.607,Z 500.485,A -85,B 0,C 180,E1 -27576.256,E2 -27576.256} C_VEL
LIN {X 0,Y 111.016,Z 505.666,A -85,B 0,C 180,E1 -27578.081,E2 -27578.081} C_VEL
LIN {X 0,Y 107.047,Z 508.518,A -85,B 0,C 180,E1 -27579.808,E2 -27579.808} C_VEL
LIN {X 0,Y 97.946,Z 515.3,A -85,B 0,C 180,E1 -27586.092,E2 -27586.092} C_VEL
LIN {X 0,Y 89.783,Z 520.823,A -85,B 0,C 180,E1 -27594.048,E2 -27594.048} C_VEL
LIN {X 0,Y 85.149,Z 523.734,A -85,B 0,C 180,E1 -27600.313,E2 -27600.313} C_VEL
LIN {X 0,Y 80.575,Z 526.567,A -85,B 0,C 180,E1 -27609.578,E2 -27609.578} C_VEL
LIN {X 0,Y 77.984,Z 528.254,A -85,B 0,C 180,E1 -27619.614,E2 -27619.614} C_VEL
LIN {X 0,Y 77.271,Z 528.833,A -85,B 0,C 180,E1 -27629.998,E2 -27629.998} C_VEL
LIN {X 0,Y 77.983,Z 528.283,A -85,B 0,C 180,E1 -27640.382,E2 -27640.382} C_VEL
LIN {X 0,Y 80.551,Z 526.635,A -85,B 0,C 180,E1 -27650.424,E2 -27650.424} C_VEL
LIN {X 0,Y 85.075,Z 523.837,A -85,B 0,C 180,E1 -27659.711,E2 -27659.711} C_VEL
LIN {X 0,Y 91.475,Z 519.812,A -85,B 0,C 180,E1 -27667.923,E2 -27667.923} C_VEL
LIN {X 0,Y 99.271,Z 514.469,A -85,B 0,C 180,E1 -27675.067,E2 -27675.067} C_VEL
LIN {X 0,Y 108.43,Z 507.635,A -85,B 0,C 180,E1 -27681.057,E2 -27681.057} C_VEL
LIN {X 0,Y 118.445,Z 499.099,A -85,B 0,C 180,E1 -27686.168,E2 -27686.168} C_VEL
LIN {X 0,Y 127.881,Z 490.006,A -85,B 0,C 180,E1 -27689.946,E2 -27689.946} C_VEL
LIN {X 0,Y 134.822,Z 482.363,A -85,B 0,C 180,E1 -27692.393,E2 -27692.393} C_VEL
LIN {X 0,Y 135.599,Z 480.493,A -85,B 0,C 180,E1 -27693.748,E2 -27693.748} C_VEL
LIN {X 0,Y 136.184,Z 475.571,A -85,B 0,C 180,E1 -27698.823,E2 -27698.823} C_VEL
LIN {X 0,Y 136.297,Z 471.977,A -85,B 0,C 180,E1 -27703.524,E2 -27703.524} C_VEL
LIN {X 0,Y 136.367,Z 469.253,A -85,B 0,C 180,E1 -27708.289,E2 -27708.289} C_VEL
LIN {X 0,Y 136.454,Z 468.007,A -85,B 0,C 180,E1 -27711.111,E2 -27711.111} C_VEL
LIN {X 0,Y 136.542,Z 467.129,A -85,B 0,C 180,E1 -27714.091,E2 -27714.091} C_VEL
LIN {X 0,Y 137.192,Z 466.136,A -85,B 0,C 180,E1 -27720,E2 -27720} C_VEL
LIN {X 0,Y 137.034,Z 466.89,A -85,B 0,C 180,E1 -27722.939,E2 -27722.939} C_VEL
LIN {X 0,Y 136.954,Z 467.99,A -85,B 0,C 180,E1 -27725.89,E2 -27725.89} C_VEL
LIN {X 0,Y 136.637,Z 470.724,A -85,B 0,C 180,E1 -27730.371,E2 -27730.371} C_VEL
LIN {X 0,Y 136.307,Z 473.273,A -85,B 0,C 180,E1 -27733.414,E2 -27733.414} C_VEL
LIN {X 0,Y 135.772,Z 476.342,A -85,B 0,C 180,E1 -27736.541,E2 -27736.541} C_VEL
LIN {X 0,Y 134.588,Z 482.095,A -85,B 0,C 180,E1 -27741.44,E2 -27741.44} C_VEL
LIN {X 0,Y 133.71,Z 485.201,A -85,B 0,C 180,E1 -27743.701,E2 -27743.701} C_VEL
LIN {X 0,Y 130.071,Z 491.521,A -85,B 0,C 180,E1 -27746.937,E2 -27746.937} C_VEL
LIN {X 0,Y 120.273,Z 501.577,A -85,B 0,C 180,E1 -27750.472,E2 -27750.472} C_VEL
LIN {X 0,Y 110.225,Z 510.635,A -85,B 0,C 180,E1 -27755.018,E2 -27755.018} C_VEL
LIN {X 0,Y 101.375,Z 517.826,A -85,B 0,C 180,E1 -27760.309,E2 -27760.309} C_VEL
LIN {X 0,Y 92.801,Z 524.108,A -85,B 0,C 180,E1 -27767.035,E2 -27767.035} C_VEL
LIN {X 0,Y 85.818,Z 528.993,A -85,B 0,C 180,E1 -27775.025,E2 -27775.025} C_VEL
LIN {X 0,Y 80.647,Z 532.592,A -85,B 0,C 180,E1 -27784.171,E2 -27784.171} C_VEL
LIN {X 0,Y 77.617,Z 534.986,A -85,B 0,C 180,E1 -27794.24,E2 -27794.24} C_VEL
LIN {X 0,Y 76.8,Z 536.22,A -85,B 0,C 180,E1 -27804.752,E2 -27804.752} C_VEL
LIN {X 0,Y 77.052,Z 536.398,A -85,B 0,C 180,E1 -27810.002,E2 -27810.002} C_VEL
LIN {X 0,Y 76.975,Z 535.727,A -85,B 0,C 180,E1 -27820.524,E2 -27820.524} C_VEL
LIN {X 0,Y 78.83,Z 533.887,A -85,B 0,C 180,E1 -27830.895,E2 -27830.895} C_VEL
LIN {X 0,Y 82.966,Z 530.876,A -85,B 0,C 180,E1 -27840.55,E2 -27840.55} C_VEL
LIN {X 0,Y 89.071,Z 526.623,A -85,B 0,C 180,E1 -27849.143,E2 -27849.143} C_VEL
LIN {X 0,Y 96.896,Z 521.025,A -85,B 0,C 180,E1 -27856.498,E2 -27856.498} C_VEL
LIN {X 0,Y 106.093,Z 513.935,A -85,B 0,C 180,E1 -27862.651,E2 -27862.651} C_VEL
LIN {X 0,Y 114.899,Z 506.364,A -85,B 0,C 180,E1 -27867.253,E2 -27867.253} C_VEL
LIN {X 0,Y 124.459,Z 497.266,A -85,B 0,C 180,E1 -27871.078,E2 -27871.078} C_VEL
LIN {X 0,Y 130.037,Z 491.259,A -85,B 0,C 180,E1 -27873.098,E2 -27873.098} C_VEL
LIN {X 0,Y 133.549,Z 485.089,A -85,B 0,C 180,E1 -27876.274,E2 -27876.274} C_VEL
LIN {X 0,Y 134.472,Z 481.936,A -85,B 0,C 180,E1 -27878.541,E2 -27878.541} C_VEL
LIN {X 0,Y 135.641,Z 476.174,A -85,B 0,C 180,E1 -27883.443,E2 -27883.443} C_VEL
LIN {X 0,Y 136.342,Z 471.744,A -85,B 0,C 180,E1 -27888.101,E2 -27888.101} C_VEL
LIN {X 0,Y 136.638,Z 469.464,A -85,B 0,C 180,E1 -27891.124,E2 -27891.124} C_VEL
LIN {X 0,Y 136.809,Z 467.799,A -85,B 0,C 180,E1 -27894.103,E2 -27894.103} C_VEL
LIN {X 0,Y 137.123,Z 465.828,A -85,B 0,C 180,E1 -27900,E2 -27900} C_VEL
LIN {X 0,Y 136.451,Z 466.845,A -85,B 0,C 180,E1 -27905.913,E2 -27905.913} C_VEL
LIN {X 0,Y 136.341,Z 467.743,A -85,B 0,C 180,E1 -27908.896,E2 -27908.896} C_VEL
LIN {X 0,Y 136.216,Z 469.119,A -85,B 0,C 180,E1 -27911.911,E2 -27911.911} C_VEL
LIN {X 0,Y 136.163,Z 470.823,A -85,B 0,C 180,E1 -27914.956,E2 -27914.956} C_VEL
LIN {X 0,Y 136.06,Z 473.942,A -85,B 0,C 180,E1 -27919.461,E2 -27919.461} C_VEL
LIN {X 0,Y 135.896,Z 476.791,A -85,B 0,C 180,E1 -27922.821,E2 -27922.821} C_VEL
LIN {X 0,Y 135.538,Z 480.129,A -85,B 0,C 180,E1 -27926.194,E2 -27926.194} C_VEL
LIN {X 0,Y 134.88,Z 482.009,A -85,B 0,C 180,E1 -27927.648,E2 -27927.648} C_VEL
LIN {X 0,Y 127.952,Z 489.683,A -85,B 0,C 180,E1 -27930.104,E2 -27930.104} C_VEL
LIN {X 0,Y 118.537,Z 498.823,A -85,B 0,C 180,E1 -27933.893,E2 -27933.893} C_VEL
LIN {X 0,Y 110.919,Z 505.418,A -85,B 0,C 180,E1 -27937.623,E2 -27937.623} C_VEL
LIN {X 0,Y 107.047,Z 508.518,A -85,B 0,C 180,E1 -27939.808,E2 -27939.808} C_VEL
LIN {X 0,Y 103.116,Z 511.25,A -85,B 0,C 180,E1 -27941.714,E2 -27941.714} C_VEL
LIN {X 0,Y 95.546,Z 515.401,A -85,B 0,C 180,E1 -27944.536,E2 -27944.536} C_VEL
LIN {X 0,Y 88.107,Z 519.037,A -85,B 0,C 180,E1 -27947.931,E2 -27947.931} C_VEL
LIN {X 0,Y 84.526,Z 520.929,A -85,B 0,C 180,E1 -27950.77,E2 -27950.77} C_VEL
LIN {X 0,Y 79.029,Z 524.084,A -85,B 0,C 180,E1 -27957.75,E2 -27957.75} C_VEL
LIN {X 0,Y 73.966,Z 526.915,A -85,B 0,C 180,E1 -27967.66,E2 -27967.66} C_VEL
LIN {X 0,Y 71.02,Z 528.602,A -85,B 0,C 180,E1 -27978.582,E2 -27978.582} C_VEL
LIN {X 0,Y 70.197,Z 529.18,A -85,B 0,C 180,E1 -27989.998,E2 -27989.998} C_VEL
LIN {X 0,Y 71.018,Z 528.631,A -85,B 0,C 180,E1 -28001.413,E2 -28001.413} C_VEL
LIN {X 0,Y 73.942,Z 526.982,A -85,B 0,C 180,E1 -28012.343,E2 -28012.343} C_VEL
LIN {X 0,Y 78.959,Z 524.186,A -85,B 0,C 180,E1 -28022.277,E2 -28022.277} C_VEL
LIN {X 0,Y 85.97,Z 520.16,A -85,B 0,C 180,E1 -28030.841,E2 -28030.841} C_VEL
LIN {X 0,Y 94.374,Z 514.817,A -85,B 0,C 180,E1 -28038.13,E2 -28038.13} C_VEL
LIN {X 0,Y 104.091,Z 507.983,A -85,B 0,C 180,E1 -28044.114,E2 -28044.114} C_VEL
LIN {X 0,Y 114.635,Z 499.446,A -85,B 0,C 180,E1 -28049.124,E2 -28049.124} C_VEL
LIN {X 0,Y 123.068,Z 491.758,A -85,B 0,C 180,E1 -28052.267,E2 -28052.267} C_VEL
LIN {X 0,Y 128.806,Z 485.866,A -85,B 0,C 180,E1 -28054.267,E2 -28054.267} C_VEL
LIN {X 0,Y 130.168,Z 484.061,A -85,B 0,C 180,E1 -28055.069,E2 -28055.069} C_VEL
LIN {X 0,Y 130.981,Z 480.037,A -85,B 0,C 180,E1 -28059.588,E2 -28059.588} C_VEL
LIN {X 0,Y 131.379,Z 476.659,A -85,B 0,C 180,E1 -28064.486,E2 -28064.486} C_VEL
LIN {X 0,Y 131.529,Z 474.946,A -85,B 0,C 180,E1 -28067.659,E2 -28067.659} C_VEL
LIN {X 0,Y 131.721,Z 473.585,A -85,B 0,C 180,E1 -28070.789,E2 -28070.789} C_VEL
LIN {X 0,Y 131.918,Z 472.656,A -85,B 0,C 180,E1 -28073.883,E2 -28073.883} C_VEL
LIN {X 0,Y 132.665,Z 471.647,A -85,B 0,C 180,E1 -28080,E2 -28080} C_VEL
LIN {X 0,Y 132.465,Z 472.441,A -85,B 0,C 180,E1 -28083.041,E2 -28083.041} C_VEL
LIN {X 0,Y 132.257,Z 473.641,A -85,B 0,C 180,E1 -28086.1,E2 -28086.1} C_VEL
LIN {X 0,Y 131.933,Z 475.394,A -85,B 0,C 180,E1 -28089.195,E2 -28089.195} C_VEL
LIN {X 0,Y 131.418,Z 477.803,A -85,B 0,C 180,E1 -28092.351,E2 -28092.351} C_VEL
LIN {X 0,Y 130.698,Z 480.792,A -85,B 0,C 180,E1 -28095.596,E2 -28095.596} C_VEL
LIN {X 0,Y 129.317,Z 485.753,A -85,B 0,C 180,E1 -28100.118,E2 -28100.118} C_VEL
LIN {X 0,Y 128.64,Z 487.723,A -85,B 0,C 180,E1 -28101.761,E2 -28101.761} C_VEL
LIN {X 0,Y 126.193,Z 491.7,A -85,B 0,C 180,E1 -28103.953,E2 -28103.953} C_VEL
LIN {X 0,Y 125.269,Z 492.963,A -85,B 0,C 180,E1 -28104.616,E2 -28104.616} C_VEL
LIN {X 0,Y 115.382,Z 502.489,A -85,B 0,C 180,E1 -28107.972,E2 -28107.972} C_VEL
LIN {X 0,Y 105.594,Z 510.808,A -85,B 0,C 180,E1 -28112.171,E2 -28112.171} C_VEL
LIN {X 0,Y 96.885,Z 517.475,A -85,B 0,C 180,E1 -28117.07,E2 -28117.07} C_VEL
LIN {X 0,Y 87.668,Z 523.756,A -85,B 0,C 180,E1 -28123.825,E2 -28123.825} C_VEL
LIN {X 0,Y 79.667,Z 528.877,A -85,B 0,C 180,E1 -28132.556,E2 -28132.556} C_VEL
LIN {X 0,Y 74.265,Z 532.242,A -85,B 0,C 180,E1 -28141.762,E2 -28141.762} C_VEL
LIN {X 0,Y 70.746,Z 534.635,A -85,B 0,C 180,E1 -28152.664,E2 -28152.664} C_VEL
LIN {X 0,Y 69.719,Z 535.871,A -85,B 0,C 180,E1 -28164.217,E2 -28164.217} C_VEL
LIN {X 0,Y 69.951,Z 536.05,A -85,B 0,C 180,E1 -28170.002,E2 -28170.002} C_VEL
LIN {X 0,Y 69.961,Z 535.377,A -85,B 0,C 180,E1 -28181.593,E2 -28181.593} C_VEL
LIN {X 0,Y 72.17,Z 533.535,A -85,B 0,C 180,E1 -28192.928,E2 -28192.928} C_VEL
LIN {X 0,Y 76.872,Z 530.523,A -85,B 0,C 180,E1 -28203.27,E2 -28203.27} C_VEL
LIN {X 0,Y 83.624,Z 526.27,A -85,B 0,C 180,E1 -28212.251,E2 -28212.251} C_VEL
LIN {X 0,Y 92.097,Z 520.672,A -85,B 0,C 180,E1 -28219.741,E2 -28219.741} C_VEL
LIN {X 0,Y 101.892,Z 513.581,A -85,B 0,C 180,E1 -28225.866,E2 -28225.866} C_VEL
LIN {X 0,Y 111.183,Z 506.011,A -85,B 0,C 180,E1 -28230.363,E2 -28230.363} C_VEL
LIN {X 0,Y 121.163,Z 496.913,A -85,B 0,C 180,E1 -28234.039,E2 -28234.039} C_VEL
LIN {X 0,Y 125.224,Z 492.753,A -85,B 0,C 180,E1 -28235.393,E2 -28235.393} C_VEL
LIN {X 0,Y 127.606,Z 489.137,A -85,B 0,C 180,E1 -28237.324,E2 -28237.324} C_VEL
LIN {X 0,Y 128.544,Z 487.441,A -85,B 0,C 180,E1 -28238.354,E2 -28238.354} C_VEL
LIN {X 0,Y 129.589,Z 484.239,A -85,B 0,C 180,E1 -28241.011,E2 -28241.011} C_VEL
LIN {X 0,Y 130.793,Z 479.77,A -85,B 0,C 180,E1 -28245.292,E2 -28245.292} C_VEL
LIN {X 0,Y 131.487,Z 476.658,A -85,B 0,C 180,E1 -28248.825,E2 -28248.825} C_VEL
LIN {X 0,Y 131.798,Z 475.212,A -85,B 0,C 180,E1 -28250.795,E2 -28250.795} C_VEL
LIN {X 0,Y 132.124,Z 473.451,A -85,B 0,C 180,E1 -28253.893,E2 -28253.893} C_VEL
LIN {X 0,Y 132.332,Z 472.235,A -85,B 0,C 180,E1 -28256.956,E2 -28256.956} C_VEL
LIN {X 0,Y 132.593,Z 471.35,A -85,B 0,C 180,E1 -28260,E2 -28260} C_VEL
LIN {X 0,Y 131.834,Z 472.385,A -85,B 0,C 180,E1 -28266.121,E2 -28266.121} C_VEL
LIN {X 0,Y 131.634,Z 473.311,A -85,B 0,C 180,E1 -28269.217,E2 -28269.217} C_VEL
LIN {X 0,Y 131.378,Z 474.739,A -85,B 0,C 180,E1 -28272.356,E2 -28272.356} C_VEL
LIN {X 0,Y 131.113,Z 477.459,A -85,B 0,C 180,E1 -28277.147,E2 -28277.147} C_VEL
LIN {X 0,Y 130.618,Z 481.261,A -85,B 0,C 180,E1 -28282.126,E2 -28282.126} C_VEL
